  MoveL 8739 to (-32.14, 37, 125.68) mm, rotated rx -180 ry 0 rz 180 deg; joints [-169.099, 67.153, -85.949, 168.501, 71.555, 3.683]
  Call Extruder(466.13359)
  MoveL 8740 to (-31.9, 36.9, 125.68) mm, rotated rx 180 ry 0 rz 180 deg; joints [-169.115, 67.132, -85.961, 168.515, 71.522, 3.684]
  MoveL 8741 to (-31.9, 36.9, 125.68) mm, rotated rx 180 ry 0 rz 180 deg; joints [-169.115, 67.132, -85.961, 168.515, 71.522, 3.684]
  Call Extruder(466.29670)
  MoveL 8742 to (-31.64, 36.79, 125.68) mm, rotated rx 180 ry 0 rz 180 deg; joints [-169.132, 67.109, -85.974, 168.531, 71.486, 3.686]
  MoveL 8743 to (-31.64, 36.79, 125.68) mm, rotated rx 180 ry 0 rz 180 deg; joints [-169.132, 67.109, -85.974, 168.531, 71.486, 3.686]
  Call Extruder(466.41015)
  MoveL 8744 to (-31.45, 36.73, 125.68) mm, rotated rx -180 ry 0 rz 180 deg; joints [-169.139, 67.093, -85.983, 168.537, 71.461, 3.689]
  MoveL 8745 to (-31.45, 36.73, 125.68) mm, rotated rx -180 ry 0 rz 180 deg; joints [-169.139, 67.093, -85.983, 168.537, 71.461, 3.689]
  Call Extruder(466.52317)
  MoveL 8746 to (-31.26, 36.67, 125.68) mm, rotated rx -180 ry 0 rz -180 deg; joints [-169.146, 67.077, -85.992, 168.543, 71.435, 3.692]
  MoveL 8747 to (-31.26, 36.67, 125.68) mm, rotated rx -180 ry 0 rz -180 deg; joints [-169.146, 67.077, -85.992, 168.543, 71.435, 3.692]
  Call Extruder(466.63573)
  MoveL 8748 to (-31.07, 36.61, 125.68) mm, rotated rx -180 ry 0 rz -180 deg; joints [-169.154, 67.06, -86.001, 168.549, 71.41, 3.695]
  MoveL 8749 to (-31.07, 36.61, 125.68) mm, rotated rx -180 ry 0 rz -180 deg; joints [-169.154, 67.06, -86.001, 168.549, 71.41, 3.695]
  Call Extruder(466.74786)
  MoveL 8750 to (-30.88, 36.55, 125.68) mm, rotated rx 180 ry 0 rz -180 deg; joints [-169.161, 67.044, -86.01, 168.555, 71.385, 3.698]
  MoveL 8751 to (-30.88, 36.55, 125.68) mm, rotated rx 180 ry 0 rz -180 deg; joints [-169.161, 67.044, -86.01, 168.555, 71.385, 3.698]
  Call Extruder(466.85954)
  MoveL 8752 to (-30.7, 36.49, 125.68) mm, rotated rx -180 ry 0 rz -180 deg; joints [-169.168, 67.028, -86.019, 168.561, 71.36, 3.701]
  MoveL 8753 to (-30.7, 36.49, 125.68) mm, rotated rx -180 ry 0 rz -180 deg; joints [-169.168, 67.028, -86.019, 168.561, 71.36, 3.701]
  Call Extruder(466.99061)
  MoveL 8754 to (-30.47, 36.42, 125.68) mm, rotated rx -180 ry 0 rz -180 deg; joints [-169.175, 67.008, -86.03, 168.566, 71.33, 3.704]
  MoveL 8755 to (-30.47, 36.42, 125.68) mm, rotated rx -180 ry 0 rz -180 deg; joints [-169.175, 67.008, -86.03, 168.566, 71.33, 3.704]
  Call Extruder(467.12112)
  MoveL 8756 to (-30.25, 36.35, 125.68) mm, rotated rx -180 ry 0 rz -180 deg; joints [-169.182, 66.989, -86.04, 168.572, 71.3, 3.708]
  MoveL 8757 to (-30.25, 36.35, 125.68) mm, rotated rx -180 ry 0 rz -180 deg; joints [-169.182, 66.989, -86.04, 168.572, 71.3, 3.708]
  Call Extruder(467.25107)
  MoveL 8758 to (-30.02, 36.28, 125.68) mm, rotated rx -180 ry 0 rz -180 deg; joints [-169.19, 66.97, -86.051, 168.577, 71.27, 3.712]
  MoveL 8759 to (-30.02, 36.28, 125.68) mm, rotated rx -180 ry 0 rz -180 deg; joints [-169.19, 66.97, -86.051, 168.577, 71.27, 3.712]
  Call Extruder(467.38045)
  MoveL 8760 to (-29.8, 36.22, 125.68) mm, rotated rx 180 ry 0 rz -180 deg; joints [-169.197, 66.95, -86.061, 168.583, 71.24, 3.716]
  MoveL 8761 to (-29.8, 36.22, 125.68) mm, rotated rx 180 ry 0 rz -180 deg; joints [-169.197, 66.95, -86.061, 168.583, 71.24, 3.716]
  Call Extruder(467.50241)
  MoveL 8762 to (-29.59, 36.16, 125.68) mm, rotated rx 180 ry 0 rz 180 deg; joints [-169.202, 66.932, -86.071, 168.586, 71.212, 3.72]
  MoveL 8763 to (-29.59, 36.16, 125.68) mm, rotated rx 180 ry 0 rz 180 deg; joints [-169.202, 66.932, -86.071, 168.586, 71.212, 3.72]
  Call Extruder(467.61726)
  MoveL 8764 to (-29.38, 36.12, 125.68) mm, rotated rx -180 ry 0 rz -180 deg; joints [-169.203, 66.915, -86.081, 168.586, 71.186, 3.725]
  MoveL 8765 to (-29.38, 36.12, 125.68) mm, rotated rx -180 ry 0 rz -180 deg; joints [-169.203, 66.915, -86.081, 168.586, 71.186, 3.725]
  Call Extruder(467.73165)
  MoveL 8766 to (-29.18, 36.07, 125.68) mm, rotated rx 180 ry 0 rz 180 deg; joints [-169.205, 66.897, -86.09, 168.586, 71.16, 3.73]
  MoveL 8767 to (-29.18, 36.07, 125.68) mm, rotated rx 180 ry 0 rz 180 deg; joints [-169.205, 66.897, -86.09, 168.586, 71.16, 3.73]
  Call Extruder(467.84560)
  MoveL 8768 to (-28.97, 36.03, 125.68) mm, rotated rx 180 ry 0 rz -180 deg; joints [-169.207, 66.88, -86.099, 168.586, 71.133, 3.735]
  MoveL 8769 to (-28.97, 36.03, 125.68) mm, rotated rx 180 ry 0 rz -180 deg; joints [-169.207, 66.88, -86.099, 168.586, 71.133, 3.735]
  Call Extruder(467.95909)
  MoveL 8770 to (-28.77, 35.98, 125.68) mm, rotated rx -180 ry 0 rz -180 deg; joints [-169.208, 66.862, -86.109, 168.586, 71.107, 3.74]
  MoveL 8771 to (-28.77, 35.98, 125.68) mm, rotated rx -180 ry 0 rz -180 deg; joints [-169.208, 66.862, -86.109, 168.586, 71.107, 3.74]
  Call Extruder(468.09637)
  MoveL 8772 to (-28.52, 35.93, 125.68) mm, rotated rx 180 ry 0 rz -180 deg; joints [-169.209, 66.841, -86.12, 168.584, 71.075, 3.747]
  MoveL 8773 to (-28.52, 35.93, 125.68) mm, rotated rx 180 ry 0 rz -180 deg; joints [-169.209, 66.841, -86.12, 168.584, 71.075, 3.747]
  Call Extruder(468.23304)
  MoveL 8774 to (-28.27, 35.88, 125.68) mm, rotated rx -180 ry 0 rz 180 deg; joints [-169.209, 66.82, -86.132, 168.582, 71.043, 3.754]
  MoveL 8775 to (-28.27, 35.88, 125.68) mm, rotated rx -180 ry 0 rz 180 deg; joints [-169.209, 66.82, -86.132, 168.582, 71.043, 3.754]
  Call Extruder(468.36910)
  MoveL 8776 to (-28.02, 35.83, 125.68) mm, rotated rx -180 ry 0 rz -180 deg; joints [-169.21, 66.798, -86.143, 168.581, 71.011, 3.76]
  MoveL 8777 to (-28.02, 35.83, 125.68) mm, rotated rx -180 ry 0 rz -180 deg; joints [-169.21, 66.798, -86.143, 168.581, 71.011, 3.76]
  Call Extruder(468.50456)
  MoveL 8778 to (-27.77, 35.78, 125.68) mm, rotated rx -180 ry 0 rz -180 deg; joints [-169.21, 66.777, -86.154, 168.579, 70.979, 3.767]
  MoveL 8779 to (-27.77, 35.78, 125.68) mm, rotated rx -180 ry 0 rz -180 deg; joints [-169.21, 66.777, -86.154, 168.579, 70.979, 3.767]
  Call Extruder(468.63940)
  MoveL 8780 to (-27.52, 35.73, 125.68) mm, rotated rx -180 ry 0 rz 180 deg; joints [-169.211, 66.756, -86.166, 168.578, 70.947, 3.773]
  MoveL 8781 to (-27.52, 35.73, 125.68) mm, rotated rx -180 ry 0 rz 180 deg; joints [-169.211, 66.756, -86.166, 168.578, 70.947, 3.773]
  Call Extruder(468.77363)
  MoveL 8782 to (-27.28, 35.68, 125.68) mm, rotated rx -180 ry 0 rz 180 deg; joints [-169.212, 66.734, -86.177, 168.576, 70.915, 3.78]
  MoveL 8783 to (-27.28, 35.68, 125.68) mm, rotated rx -180 ry 0 rz 180 deg; joints [-169.212, 66.734, -86.177, 168.576, 70.915, 3.78]
  Call Extruder(468.90725)
  MoveL 8784 to (-27.03, 35.63, 125.68) mm, rotated rx 180 ry 0 rz 180 deg; joints [-169.212, 66.713, -86.188, 168.575, 70.883, 3.787]
  MoveL 8785 to (-27.03, 35.63, 125.68) mm, rotated rx 180 ry 0 rz 180 deg; joints [-169.212, 66.713, -86.188, 168.575, 70.883, 3.787]
  Call Extruder(469.06935)
  MoveL 8786 to (-26.72, 35.59, 125.68) mm, rotated rx 180 ry 0 rz 180 deg; joints [-169.21, 66.687, -86.202, 168.569, 70.844, 3.796]
  MoveL 8787 to (-26.72, 35.59, 125.68) mm, rotated rx 180 ry 0 rz 180 deg; joints [-169.21, 66.687, -86.202, 168.569, 70.844, 3.796]
  Call Extruder(469.23072)
  MoveL 8788 to (-26.41, 35.54, 125.68) mm, rotated rx -180 ry 0 rz 180 deg; joints [-169.207, 66.661, -86.215, 168.563, 70.805, 3.805]
  MoveL 8789 to (-26.41, 35.54, 125.68) mm, rotated rx -180 ry 0 rz 180 deg; joints [-169.207, 66.661, -86.215, 168.563, 70.805, 3.805]
  Call Extruder(469.39136)
  MoveL 8790 to (-26.11, 35.49, 125.68) mm, rotated rx 180 ry 0 rz 180 deg; joints [-169.204, 66.635, -86.229, 168.557, 70.767, 3.815]
  MoveL 8791 to (-26.11, 35.49, 125.68) mm, rotated rx 180 ry 0 rz 180 deg; joints [-169.204, 66.635, -86.229, 168.557, 70.767, 3.815]
  Call Extruder(469.55127)
  MoveL 8792 to (-25.8, 35.44, 125.68) mm, rotated rx 180 ry 0 rz 180 deg; joints [-169.201, 66.609, -86.242, 168.551, 70.728, 3.824]
  MoveL 8793 to (-25.8, 35.44, 125.68) mm, rotated rx 180 ry 0 rz 180 deg; joints [-169.201, 66.609, -86.242, 168.551, 70.728, 3.824]
  Call Extruder(469.71046)
  MoveL 8794 to (-25.5, 35.39, 125.68) mm, rotated rx -180 ry 0 rz -180 deg; joints [-169.198, 66.582, -86.256, 168.546, 70.689, 3.833]
  MoveL 8795 to (-25.5, 35.39, 125.68) mm, rotated rx -180 ry 0 rz -180 deg; joints [-169.198, 66.582, -86.256, 168.546, 70.689, 3.833]
  Call Extruder(469.86892)
  MoveL 8796 to (-25.19, 35.34, 125.68) mm, rotated rx -180 ry 0 rz -180 deg; joints [-169.195, 66.556, -86.269, 168.54, 70.65, 3.843]
  MoveL 8797 to (-25.19, 35.34, 125.68) mm, rotated rx -180 ry 0 rz -180 deg; joints [-169.195, 66.556, -86.269, 168.54, 70.65, 3.843]
  Call Extruder(470.06779)
  MoveL 8798 to (-24.8, 35.3, 125.68) mm, rotated rx 180 ry 0 rz 180 deg; joints [-169.187, 66.523, -86.286, 168.527, 70.602, 3.856]
  MoveL 8799 to (-24.8, 35.3, 125.68) mm, rotated rx 180 ry 0 rz 180 deg; joints [-169.187, 66.523, -86.286, 168.527, 70.602, 3.856]
  Call Extruder(470.26580)
  MoveL 8800 to (-24.42, 35.25, 125.68) mm, rotated rx -180 ry 0 rz -180 deg; joints [-169.178, 66.49, -86.303, 168.515, 70.554, 3.87]
  MoveL 8801 to (-24.42, 35.25, 125.68) mm, rotated rx -180 ry 0 rz -180 deg; joints [-169.178, 66.49, -86.303, 168.515, 70.554, 3.87]
  Call Extruder(470.46294)
  MoveL 8802 to (-24.03, 35.21, 125.68) mm, rotated rx -180 ry 0 rz -180 deg; joints [-169.17, 66.457, -86.32, 168.502, 70.506, 3.883]
  MoveL 8803 to (-24.03, 35.21, 125.68) mm, rotated rx -180 ry 0 rz -180 deg; joints [-169.17, 66.457, -86.32, 168.502, 70.506, 3.883]
  Call Extruder(470.65922)
  MoveL 8804 to (-23.64, 35.16, 125.68) mm, rotated rx -180 ry 0 rz 180 deg; joints [-169.161, 66.424, -86.337, 168.49, 70.457, 3.897]
  MoveL 8805 to (-23.64, 35.16, 125.68) mm, rotated rx -180 ry 0 rz 180 deg; joints [-169.161, 66.424, -86.337, 168.49, 70.457, 3.897]
  Call Extruder(470.90490)
  MoveL 8806 to (-23.15, 35.11, 125.68) mm, rotated rx 180 ry 0 rz 180 deg; joints [-169.147, 66.382, -86.357, 168.47, 70.397, 3.915]
  MoveL 8807 to (-23.15, 35.11, 125.68) mm, rotated rx 180 ry 0 rz 180 deg; joints [-169.147, 66.382, -86.357, 168.47, 70.397, 3.915]
  Call Extruder(471.19963)
  MoveL 8808 to (-22.56, 35.07, 125.68) mm, rotated rx 180 ry 0 rz 180 deg; joints [-169.127, 66.332, -86.382, 168.444, 70.325, 3.938]
  MoveL 8809 to (-22.56, 35.07, 125.68) mm, rotated rx 180 ry 0 rz 180 deg; joints [-169.127, 66.332, -86.382, 168.444, 70.325, 3.938]
  Call Extruder(471.49303)
  MoveL 8810 to (-21.97, 35.02, 125.68) mm, rotated rx -180 ry 0 rz -180 deg; joints [-169.107, 66.282, -86.407, 168.417, 70.252, 3.962]
  MoveL 8811 to (-21.97, 35.02, 125.68) mm, rotated rx -180 ry 0 rz -180 deg; joints [-169.107, 66.282, -86.407, 168.417, 70.252, 3.962]
  Call Extruder(471.92636)
  MoveL 8812 to (-21.1, 34.98, 125.68) mm, rotated rx 180 ry 0 rz -180 deg; joints [-169.069, 66.207, -86.444, 168.369, 70.146, 3.999]
  MoveL 8813 to (-21.1, 34.98, 125.68) mm, rotated rx 180 ry 0 rz -180 deg; joints [-169.069, 66.207, -86.444, 168.369, 70.146, 3.999]
  Call Extruder(472.49852)
  MoveL 8814 to (-19.94, 34.93, 125.68) mm, rotated rx -180 ry 0 rz -180 deg; joints [-169.014, 66.108, -86.492, 168.3, 70.006, 4.05]
  MoveL 8815 to (-19.94, 34.93, 125.68) mm, rotated rx -180 ry 0 rz -180 deg; joints [-169.014, 66.108, -86.492, 168.3, 70.006, 4.05]
  Call Extruder(472.92635)
  MoveL 8816 to (-19.06, 34.91, 125.68) mm, rotated rx -180 ry 0 rz -180 deg; joints [-168.967, 66.034, -86.527, 168.242, 69.901, 4.091]
  Call Extruder(589.57504)
  MoveL 8817 to (219.06, 34.91, 125.68) mm, rotated rx -180 ry 0 rz 180 deg; joints [-30.588, 54.353, -88.738, 35.613, 119.089, 19.2]
  MoveL 8818 to (219.06, 34.91, 125.68) mm, rotated rx -180 ry 0 rz 180 deg; joints [-30.588, 54.353, -88.738, 35.613, 119.089, 19.2]
  Call Extruder(590.29061)
  MoveL 8819 to (220.52, 34.95, 125.68) mm, rotated rx -180 ry 0 rz 180 deg; joints [-30.009, 54.502, -88.741, 34.939, 119.158, 18.798]
  MoveL 8820 to (220.52, 34.95, 125.68) mm, rotated rx -180 ry 0 rz 180 deg; joints [-30.009, 54.502, -88.741, 34.939, 119.158, 18.798]
  Call Extruder(590.86535)
  MoveL 8821 to (221.68, 35, 125.68) mm, rotated rx -180 ry 0 rz 180 deg; joints [-29.572, 54.622, -88.743, 34.427, 119.201, 18.489]
  MoveL 8822 to (221.68, 35, 125.68) mm, rotated rx -180 ry 0 rz 180 deg; joints [-29.572, 54.622, -88.743, 34.427, 119.201, 18.489]
  Call Extruder(591.15874)
  MoveL 8823 to (222.27, 35.05, 125.68) mm, rotated rx -180 ry 0 rz 180 deg; joints [-29.371, 54.685, -88.744, 34.19, 119.213, 18.343]
  MoveL 8824 to (222.27, 35.05, 125.68) mm, rotated rx -180 ry 0 rz 180 deg; joints [-29.371, 54.685, -88.744, 34.19, 119.213, 18.343]
  Call Extruder(591.45347)
  MoveL 8825 to (222.86, 35.09, 125.68) mm, rotated rx -180 ry 0 rz 180 deg; joints [-29.173, 54.747, -88.744, 33.955, 119.224, 18.198]
  MoveL 8826 to (222.86, 35.09, 125.68) mm, rotated rx -180 ry 0 rz 180 deg; joints [-29.173, 54.747, -88.744, 33.955, 119.224, 18.198]
  Call Extruder(591.74952)
  MoveL 8827 to (223.45, 35.14, 125.68) mm, rotated rx -180 ry 0 rz 180 deg; joints [-28.978, 54.809, -88.745, 33.723, 119.233, 18.055]
  MoveL 8828 to (223.45, 35.14, 125.68) mm, rotated rx -180 ry 0 rz 180 deg; joints [-28.978, 54.809, -88.745, 33.723, 119.233, 18.055]
  Call Extruder(591.94580)
  MoveL 8829 to (223.83, 35.18, 125.68) mm, rotated rx -180 ry 0 rz 180 deg; joints [-28.862, 54.851, -88.745, 33.584, 119.235, 17.967]
  MoveL 8830 to (223.83, 35.18, 125.68) mm, rotated rx -180 ry 0 rz 180 deg; joints [-28.862, 54.851, -88.745, 33.584, 119.235, 17.967]
  Call Extruder(592.14294)
  MoveL 8831 to (224.22, 35.23, 125.68) mm, rotated rx -180 ry 0 rz 180 deg; joints [-28.747, 54.893, -88.745, 33.445, 119.235, 17.879]
  MoveL 8832 to (224.22, 35.23, 125.68) mm, rotated rx -180 ry 0 rz 180 deg; joints [-28.747, 54.893, -88.745, 33.445, 119.235, 17.879]
  Call Extruder(592.34095)
  MoveL 8833 to (224.61, 35.27, 125.68) mm, rotated rx -180 ry 0 rz 180 deg; joints [-28.633, 54.935, -88.746, 33.309, 119.235, 17.793]
  MoveL 8834 to (224.61, 35.27, 125.68) mm, rotated rx -180 ry 0 rz 180 deg; joints [-28.633, 54.935, -88.746, 33.309, 119.235, 17.793]
  Call Extruder(592.53982)
  MoveL 8835 to (225, 35.32, 125.68) mm, rotated rx 180 ry 0 rz 180 deg; joints [-28.52, 54.977, -88.746, 33.173, 119.235, 17.706]
  MoveL 8836 to (225, 35.32, 125.68) mm, rotated rx 180 ry 0 rz 180 deg; joints [-28.52, 54.977, -88.746, 33.173, 119.235, 17.706]
  Call Extruder(592.71890)
  MoveL 8837 to (225.34, 35.37, 125.68) mm, rotated rx -180 ry 0 rz 180 deg; joints [-28.425, 55.015, -88.746, 33.057, 119.232, 17.632]
  MoveL 8838 to (225.34, 35.37, 125.68) mm, rotated rx -180 ry 0 rz 180 deg; joints [-28.425, 55.015, -88.746, 33.057, 119.232, 17.632]
  Call Extruder(592.87809)
  MoveL 8839 to (225.65, 35.42, 125.68) mm, rotated rx 180 ry 0 rz 180 deg; joints [-28.346, 55.049, -88.746, 32.961, 119.228, 17.569]
  MoveL 8840 to (225.65, 35.42, 125.68) mm, rotated rx 180 ry 0 rz 180 deg; joints [-28.346, 55.049, -88.746, 32.961, 119.228, 17.569]
  Call Extruder(593.03800)
  MoveL 8841 to (225.96, 35.47, 125.68) mm, rotated rx -180 ry 0 rz 180 deg; joints [-28.267, 55.082, -88.746, 32.864, 119.223, 17.506]
  MoveL 8842 to (225.96, 35.47, 125.68) mm, rotated rx -180 ry 0 rz 180 deg; joints [-28.267, 55.082, -88.746, 32.864, 119.223, 17.506]
  Call Extruder(593.19864)
  MoveL 8843 to (226.26, 35.51, 125.68) mm, rotated rx -180 ry 0 rz 180 deg; joints [-28.19, 55.116, -88.746, 32.77, 119.218, 17.443]
  MoveL 8844 to (226.26, 35.51, 125.68) mm, rotated rx -180 ry 0 rz 180 deg; joints [-28.19, 55.116, -88.746, 32.77, 119.218, 17.443]
  Call Extruder(593.36001)
  MoveL 8845 to (226.57, 35.56, 125.68) mm, rotated rx -180 ry 0 rz -180 deg; joints [-28.112, 55.15, -88.746, 32.675, 119.213, 17.381]
  MoveL 8846 to (226.57, 35.56, 125.68) mm, rotated rx -180 ry 0 rz -180 deg; joints [-28.112, 55.15, -88.746, 32.675, 119.213, 17.381]
  Call Extruder(593.52210)
  MoveL 8847 to (226.87, 35.61, 125.68) mm, rotated rx -180 ry 0 rz 180 deg; joints [-28.036, 55.184, -88.746, 32.581, 119.207, 17.319]
  MoveL 8848 to (226.87, 35.61, 125.68) mm, rotated rx -180 ry 0 rz 180 deg; joints [-28.036, 55.184, -88.746, 32.581, 119.207, 17.319]
  Call Extruder(593.67030)
  MoveL 8849 to (227.15, 35.66, 125.68) mm, rotated rx 180 ry 0 rz 180 deg; joints [-27.971, 55.215, -88.746, 32.5, 119.2, 17.265]
  MoveL 8850 to (227.15, 35.66, 125.68) mm, rotated rx 180 ry 0 rz 180 deg; joints [-27.971, 55.215, -88.746, 32.5, 119.2, 17.265]
  Call Extruder(593.80453)
  MoveL 8851 to (227.4, 35.71, 125.68) mm, rotated rx -180 ry 0 rz 180 deg; joints [-27.915, 55.243, -88.746, 32.431, 119.193, 17.219]
  MoveL 8852 to (227.4, 35.71, 125.68) mm, rotated rx -180 ry 0 rz 180 deg; joints [-27.915, 55.243, -88.746, 32.431, 119.193, 17.219]
  Call Extruder(593.93938)
  MoveL 8853 to (227.65, 35.76, 125.68) mm, rotated rx -180 ry 0 rz -180 deg; joints [-27.861, 55.271, -88.746, 32.363, 119.185, 17.172]
  MoveL 8854 to (227.65, 35.76, 125.68) mm, rotated rx -180 ry 0 rz -180 deg; joints [-27.861, 55.271, -88.746, 32.363, 119.185, 17.172]
  Call Extruder(594.07483)
  MoveL 8855 to (227.9, 35.81, 125.68) mm, rotated rx -180 ry 0 rz 180 deg; joints [-27.807, 55.299, -88.745, 32.295, 119.178, 17.126]
  MoveL 8856 to (227.9, 35.81, 125.68) mm, rotated rx -180 ry 0 rz 180 deg; joints [-27.807, 55.299, -88.745, 32.295, 119.178, 17.126]
  Call Extruder(594.21089)
  MoveL 8857 to (228.15, 35.86, 125.68) mm, rotated rx 180 ry 0 rz 180 deg; joints [-27.753, 55.327, -88.745, 32.228, 119.169, 17.08]
  MoveL 8858 to (228.15, 35.86, 125.68) mm, rotated rx 180 ry 0 rz 180 deg; joints [-27.753, 55.327, -88.745, 32.228, 119.169, 17.08]
  Call Extruder(594.34757)
  MoveL 8859 to (228.4, 35.91, 125.68) mm, rotated rx 180 ry 0 rz 180 deg; joints [-27.699, 55.355, -88.745, 32.161, 119.161, 17.034]
  MoveL 8860 to (228.4, 35.91, 125.68) mm, rotated rx 180 ry 0 rz 180 deg; joints [-27.699, 55.355, -88.745, 32.161, 119.161, 17.034]
  Call Extruder(594.48485)
  MoveL 8861 to (228.64, 35.96, 125.68) mm, rotated rx -180 ry 0 rz -180 deg; joints [-27.646, 55.383, -88.745, 32.094, 119.153, 16.989]
  MoveL 8862 to (228.64, 35.96, 125.68) mm, rotated rx -180 ry 0 rz -180 deg; joints [-27.646, 55.383, -88.745, 32.094, 119.153, 16.989]
  Call Extruder(594.61052)
  MoveL 8863 to (228.87, 36, 125.68) mm, rotated rx 180 ry 0 rz 180 deg; joints [-27.599, 55.408, -88.745, 32.036, 119.145, 16.948]
  MoveL 8864 to (228.87, 36, 125.68) mm, rotated rx 180 ry 0 rz 180 deg; joints [-27.599, 55.408, -88.745, 32.036, 119.145, 16.948]
  Call Extruder(594.72447)
  MoveL 8865 to (229.08, 36.05, 125.68) mm, rotated rx -180 ry 0 rz 180 deg; joints [-27.559, 55.431, -88.744, 31.984, 119.137, 16.912]
  MoveL 8866 to (229.08, 36.05, 125.68) mm, rotated rx -180 ry 0 rz 180 deg; joints [-27.559, 55.431, -88.744, 31.984, 119.137, 16.912]
  Call Extruder(594.83887)
  MoveL 8867 to (229.28, 36.09, 125.68) mm, rotated rx -180 ry 0 rz 180 deg; joints [-27.518, 55.455, -88.744, 31.933, 119.129, 16.877]
  MoveL 8868 to (229.28, 36.09, 125.68) mm, rotated rx -180 ry 0 rz 180 deg; joints [-27.518, 55.455, -88.744, 31.933, 119.129, 16.877]
  Call Extruder(594.95372)
  MoveL 8869 to (229.48, 36.14, 125.68) mm, rotated rx -180 ry 0 rz 180 deg; joints [-27.479, 55.478, -88.744, 31.882, 119.12, 16.841]
  MoveL 8870 to (229.48, 36.14, 125.68) mm, rotated rx -180 ry 0 rz 180 deg; joints [-27.479, 55.478, -88.744, 31.882, 119.12, 16.841]
  Call Extruder(595.06902)
  MoveL 8871 to (229.69, 36.18, 125.68) mm, rotated rx -180 ry 0 rz 180 deg; joints [-27.439, 55.501, -88.744, 31.832, 119.112, 16.806]
  MoveL 8872 to (229.69, 36.18, 125.68) mm, rotated rx -180 ry 0 rz 180 deg; joints [-27.439, 55.501, -88.744, 31.832, 119.112, 16.806]
  Call Extruder(595.20041)
  MoveL 8873 to (229.92, 36.25, 125.68) mm, rotated rx -180 ry 0 rz 180 deg; joints [-27.404, 55.528, -88.743, 31.786, 119.099, 16.771]
  MoveL 8874 to (229.92, 36.25, 125.68) mm, rotated rx -180 ry 0 rz 180 deg; joints [-27.404, 55.528, -88.743, 31.786, 119.099, 16.771]
  Call Extruder(595.31352)
  MoveL 8875 to (230.11, 36.31, 125.68) mm, rotated rx -180 ry 0 rz 180 deg; joints [-27.377, 55.55, -88.743, 31.75, 119.087, 16.743]
  MoveL 8876 to (230.11, 36.31, 125.68) mm, rotated rx -180 ry 0 rz 180 deg; joints [-27.377, 55.55, -88.743, 31.75, 119.087, 16.743]
  Call Extruder(595.42707)
  MoveL 8877 to (230.31, 36.37, 125.68) mm, rotated rx -180 ry 0 rz 180 deg; joints [-27.351, 55.573, -88.743, 31.714, 119.075, 16.715]
  MoveL 8878 to (230.31, 36.37, 125.68) mm, rotated rx -180 ry 0 rz 180 deg; joints [-27.351, 55.573, -88.743, 31.714, 119.075, 16.715]
  Call Extruder(595.54106)
  MoveL 8879 to (230.5, 36.43, 125.68) mm, rotated rx -180 ry 0 rz 180 deg; joints [-27.325, 55.596, -88.742, 31.679, 119.062, 16.687]
  MoveL 8880 to (230.5, 36.43, 125.68) mm, rotated rx -180 ry 0 rz 180 deg; joints [-27.325, 55.596, -88.742, 31.679, 119.062, 16.687]
  Call Extruder(595.65549)
  MoveL 8881 to (230.7, 36.49, 125.68) mm, rotated rx -180 ry 0 rz 180 deg; joints [-27.299, 55.619, -88.742, 31.644, 119.05, 16.659]
  MoveL 8882 to (230.7, 36.49, 125.68) mm, rotated rx -180 ry 0 rz 180 deg; joints [-27.299, 55.619, -88.742, 31.644, 119.05, 16.659]
  Call Extruder(595.76739)
  MoveL 8883 to (230.88, 36.55, 125.68) mm, rotated rx 180 ry 0 rz 180 deg; joints [-27.276, 55.642, -88.742, 31.612, 119.037, 16.633]
  MoveL 8884 to (230.88, 36.55, 125.68) mm, rotated rx 180 ry 0 rz 180 deg; joints [-27.276, 55.642, -88.742, 31.612, 119.037, 16.633]
  Call Extruder(595.87973)
  MoveL 8885 to (231.07, 36.61, 125.68) mm, rotated rx -180 ry 0 rz 180 deg; joints [-27.253, 55.664, -88.741, 31.58, 119.025, 16.607]
  MoveL 8886 to (231.07, 36.61, 125.68) mm, rotated rx -180 ry 0 rz 180 deg; joints [-27.253, 55.664, -88.741, 31.58, 119.025, 16.607]
  Call Extruder(595.99252)
  MoveL 8887 to (231.26, 36.67, 125.68) mm, rotated rx -180 ry 0 rz -180 deg; joints [-27.231, 55.686, -88.741, 31.549, 119.012, 16.582]
  MoveL 8888 to (231.26, 36.67, 125.68) mm, rotated rx -180 ry 0 rz -180 deg; joints [-27.231, 55.686, -88.741, 31.549, 119.012, 16.582]
  Call Extruder(596.10575)
  MoveL 8889 to (231.45, 36.73, 125.68) mm, rotated rx -180 ry 0 rz 180 deg; joints [-27.208, 55.709, -88.74, 31.517, 118.999, 16.556]
  MoveL 8890 to (231.45, 36.73, 125.68) mm, rotated rx -180 ry 0 rz 180 deg; joints [-27.208, 55.709, -88.74, 31.517, 118.999, 16.556]
  Call Extruder(596.21943)
  MoveL 8891 to (231.64, 36.79, 125.68) mm, rotated rx -180 ry 0 rz 180 deg; joints [-27.185, 55.731, -88.74, 31.486, 118.986, 16.531]
  MoveL 8892 to (231.64, 36.79, 125.68) mm, rotated rx -180 ry 0 rz 180 deg; joints [-27.185, 55.731, -88.74, 31.486, 118.986, 16.531]
  Call Extruder(596.40139)
  MoveL 8893 to (231.93, 36.91, 125.68) mm, rotated rx -180 ry 0 rz 180 deg; joints [-27.167, 55.767, -88.739, 31.455, 118.96, 16.499]
  MoveL 8894 to (231.93, 36.91, 125.68) mm, rotated rx -180 ry 0 rz 180 deg; joints [-27.167, 55.767, -88.739, 31.455, 118.96, 16.499]
  Call Extruder(596.58411)
  MoveL 8895 to (232.22, 37.04, 125.68) mm, rotated rx 180 ry 0 rz -180 deg; joints [-27.149, 55.803, -88.739, 31.425, 118.933, 16.468]
  MoveL 8896 to (232.22, 37.04, 125.68) mm, rotated rx 180 ry 0 rz -180 deg; joints [-27.149, 55.803, -88.739, 31.425, 118.933, 16.468]
  Call Extruder(596.75452)
  MoveL 8897 to (232.49, 37.15, 125.68) mm, rotated rx 180 ry 0 rz 180 deg; joints [-27.133, 55.836, -88.738, 31.398, 118.909, 16.439]
  MoveL 8898 to (232.49, 37.15, 125.68) mm, rotated rx 180 ry 0 rz 180 deg; joints [-27.133, 55.836, -88.738, 31.398, 118.909, 16.439]
  Call Extruder(596.91252)
  MoveL 8899 to (232.74, 37.26, 125.68) mm, rotated rx 180 ry 0 rz 180 deg; joints [-27.121, 55.867, -88.737, 31.375, 118.885, 16.414]
  MoveL 8900 to (232.74, 37.26, 125.68) mm, rotated rx 180 ry 0 rz 180 deg; joints [-27.121, 55.867, -88.737, 31.375, 118.885, 16.414]
  Call Extruder(597.07112)
  MoveL 8901 to (232.99, 37.36, 125.68) mm, rotated rx -180 ry 0 rz -180 deg; joints [-27.108, 55.898, -88.737, 31.352, 118.862, 16.388]
  MoveL 8902 to (232.99, 37.36, 125.68) mm, rotated rx -180 ry 0 rz -180 deg; joints [-27.108, 55.898, -88.737, 31.352, 118.862, 16.388]
  Call Extruder(597.27729)
  MoveL 8903 to (233.29, 37.54, 125.68) mm, rotated rx 180 ry 0 rz 180 deg; joints [-27.12, 55.938, -88.736, 31.353, 118.824, 16.37]
  MoveL 8904 to (233.29, 37.54, 125.68) mm, rotated rx 180 ry 0 rz 180 deg; joints [-27.12, 55.938, -88.736, 31.353, 118.824, 16.37]
  Call Extruder(597.48423)
  MoveL 8905 to (233.6, 37.71, 125.68) mm, rotated rx 180 ry 0 rz -180 deg; joints [-27.132, 55.978, -88.735, 31.355, 118.785, 16.352]
  MoveL 8906 to (233.6, 37.71, 125.68) mm, rotated rx 180 ry 0 rz -180 deg; joints [-27.132, 55.978, -88.735, 31.355, 118.785, 16.352]
  Call Extruder(597.69196)
  MoveL 8907 to (233.9, 37.89, 125.68) mm, rotated rx 180 ry 0 rz 180 deg; joints [-27.144, 56.018, -88.733, 31.356, 118.747, 16.334]
  MoveL 8908 to (233.9, 37.89, 125.68) mm, rotated rx 180 ry 0 rz 180 deg; joints [-27.144, 56.018, -88.733, 31.356, 118.747, 16.334]
  Call Extruder(597.90046)
  MoveL 8909 to (234.21, 38.07, 125.68) mm, rotated rx -180 ry 0 rz 180 deg; joints [-27.156, 56.058, -88.732, 31.358, 118.709, 16.316]
  MoveL 8910 to (234.21, 38.07, 125.68) mm, rotated rx -180 ry 0 rz 180 deg; joints [-27.156, 56.058, -88.732, 31.358, 118.709, 16.316]
  Call Extruder(598.08001)
  MoveL 8911 to (234.45, 38.24, 125.68) mm, rotated rx -180 ry 0 rz 180 deg; joints [-27.187, 56.092, -88.731, 31.382, 118.67, 16.312]
  MoveL 8912 to (234.45, 38.24, 125.68) mm, rotated rx -180 ry 0 rz 180 deg; joints [-27.187, 56.092, -88.731, 31.382, 118.67, 16.312]
  Call Extruder(598.41342)
  MoveL 8913 to (234.9, 38.57, 125.68) mm, rotated rx 180 ry 0 rz 180 deg; joints [-27.245, 56.154, -88.729, 31.427, 118.599, 16.304]
  MoveL 8914 to (234.9, 38.57, 125.68) mm, rotated rx 180 ry 0 rz 180 deg; joints [-27.245, 56.154, -88.729, 31.427, 118.599, 16.304]
  Call Extruder(598.74802)
  MoveL 8915 to (235.35, 38.9, 125.68) mm, rotated rx -180 ry 0 rz 180 deg; joints [-27.302, 56.217, -88.727, 31.471, 118.528, 16.296]
  Call Extruder(599.57597)
  MoveL 8916 to (236.39, 39.81, 125.68) mm, rotated rx 180 ry 0 rz 180 deg; joints [-27.525, 56.368, -88.722, 31.67, 118.332, 16.318]
  Call Extruder(600.40391)
  MoveL 8917 to (237.3, 40.85, 125.68) mm, rotated rx -180 ry 0 rz 180 deg; joints [-27.851, 56.514, -88.716, 31.983, 118.111, 16.395]
  Call Extruder(600.57121)
  MoveL 8918 to (237.47, 41.07, 125.68) mm, rotated rx 180 ry 0 rz 180 deg; joints [-27.932, 56.542, -88.715, 32.062, 118.063, 16.419]
  MoveL 8919 to (237.47, 41.07, 125.68) mm, rotated rx 180 ry 0 rz 180 deg; joints [-27.932, 56.542, -88.715, 32.062, 118.063, 16.419]
  Call Extruder(600.90463)
  MoveL 8920 to (237.79, 41.52, 125.68) mm, rotated rx 180 ry 0 rz -180 deg; joints [-28.091, 56.598, -88.712, 32.218, 117.968, 16.465]
  MoveL 8921 to (237.79, 41.52, 125.68) mm, rotated rx 180 ry 0 rz -180 deg; joints [-28.091, 56.598, -88.712, 32.218, 117.968, 16.465]
  Call Extruder(601.23686)
  MoveL 8922 to (238.12, 41.98, 125.68) mm, rotated rx -180 ry 0 rz -180 deg; joints [-28.249, 56.655, -88.71, 32.372, 117.874, 16.509]
  MoveL 8923 to (238.12, 41.98, 125.68) mm, rotated rx -180 ry 0 rz -180 deg; joints [-28.249, 56.655, -88.71, 32.372, 117.874, 16.509]
  Call Extruder(601.35455)
  MoveL 8924 to (238.22, 42.15, 125.68) mm, rotated rx -180 ry 0 rz 180 deg; joints [-28.315, 56.674, -88.709, 32.439, 117.838, 16.531]
  MoveL 8925 to (238.22, 42.15, 125.68) mm, rotated rx -180 ry 0 rz 180 deg; joints [-28.315, 56.674, -88.709, 32.439, 117.838, 16.531]
  Call Extruder(601.56228)
  MoveL 8926 to (238.4, 42.45, 125.68) mm, rotated rx -180 ry 0 rz 180 deg; joints [-28.434, 56.707, -88.707, 32.557, 117.775, 16.569]
  MoveL 8927 to (238.4, 42.45, 125.68) mm, rotated rx -180 ry 0 rz 180 deg; joints [-28.434, 56.707, -88.707, 32.557, 117.775, 16.569]
  Call Extruder(601.76922)
  MoveL 8928 to (238.57, 42.75, 125.68) mm, rotated rx -180 ry 0 rz 180 deg; joints [-28.552, 56.741, -88.706, 32.675, 117.711, 16.607]
  MoveL 8929 to (238.57, 42.75, 125.68) mm, rotated rx -180 ry 0 rz 180 deg; joints [-28.552, 56.741, -88.706, 32.675, 117.711, 16.607]
  Call Extruder(601.97539)
  MoveL 8930 to (238.75, 43.06, 125.68) mm, rotated rx 180 ry 0 rz 180 deg; joints [-28.669, 56.774, -88.704, 32.792, 117.648, 16.644]
  MoveL 8931 to (238.75, 43.06, 125.68) mm, rotated rx 180 ry 0 rz 180 deg; joints [-28.669, 56.774, -88.704, 32.792, 117.648, 16.644]
  Call Extruder(602.15708)
  MoveL 8932 to (238.89, 43.33, 125.68) mm, rotated rx -180 ry 0 rz 180 deg; joints [-28.78, 56.803, -88.703, 32.903, 117.591, 16.682]
  MoveL 8933 to (238.89, 43.33, 125.68) mm, rotated rx -180 ry 0 rz 180 deg; joints [-28.78, 56.803, -88.703, 32.903, 117.591, 16.682]
  Call Extruder(602.31509)
  MoveL 8934 to (239, 43.58, 125.68) mm, rotated rx -180 ry 0 rz -180 deg; joints [-28.886, 56.827, -88.701, 33.011, 117.539, 16.719]
  MoveL 8935 to (239, 43.58, 125.68) mm, rotated rx -180 ry 0 rz -180 deg; joints [-28.886, 56.827, -88.701, 33.011, 117.539, 16.719]
  Call Extruder(602.47250)
  MoveL 8936 to (239.1, 43.83, 125.68) mm, rotated rx -180 ry 0 rz 180 deg; joints [-28.991, 56.851, -88.7, 33.117, 117.488, 16.756]
  MoveL 8937 to (239.1, 43.83, 125.68) mm, rotated rx -180 ry 0 rz 180 deg; joints [-28.991, 56.851, -88.7, 33.117, 117.488, 16.756]
  Call Extruder(602.65521)
  MoveL 8938 to (239.23, 44.12, 125.68) mm, rotated rx -180 ry 0 rz 180 deg; joints [-29.116, 56.879, -88.699, 33.244, 117.427, 16.8]
  MoveL 8939 to (239.23, 44.12, 125.68) mm, rotated rx -180 ry 0 rz 180 deg; joints [-29.116, 56.879, -88.699, 33.244, 117.427, 16.8]
  Call Extruder(602.83717)
  MoveL 8940 to (239.35, 44.42, 125.68) mm, rotated rx 180 ry 0 rz 180 deg; joints [-29.24, 56.907, -88.697, 33.369, 117.367, 16.844]
  MoveL 8941 to (239.35, 44.42, 125.68) mm, rotated rx 180 ry 0 rz 180 deg; joints [-29.24, 56.907, -88.697, 33.369, 117.367, 16.844]
  Call Extruder(602.98450)
  MoveL 8942 to (239.44, 44.66, 125.68) mm, rotated rx -180 ry 0 rz -180 deg; joints [-29.343, 56.929, -88.696, 33.474, 117.318, 16.88]
  MoveL 8943 to (239.44, 44.66, 125.68) mm, rotated rx -180 ry 0 rz -180 deg; joints [-29.343, 56.929, -88.696, 33.474, 117.318, 16.88]
  Call Extruder(603.09774)
  MoveL 8944 to (239.5, 44.85, 125.68) mm, rotated rx -180 ry 0 rz 180 deg; joints [-29.428, 56.945, -88.695, 33.56, 117.279, 16.911]
  MoveL 8945 to (239.5, 44.85, 125.68) mm, rotated rx -180 ry 0 rz 180 deg; joints [-29.428, 56.945, -88.695, 33.56, 117.279, 16.911]
  Call Extruder(603.21053)
  MoveL 8946 to (239.56, 45.03, 125.68) mm, rotated rx -180 ry 0 rz -180 deg; joints [-29.512, 56.961, -88.694, 33.645, 117.24, 16.942]
  MoveL 8947 to (239.56, 45.03, 125.68) mm, rotated rx -180 ry 0 rz -180 deg; joints [-29.512, 56.961, -88.694, 33.645, 117.24, 16.942]
  Call Extruder(603.32287)
  MoveL 8948 to (239.62, 45.22, 125.68) mm, rotated rx -180 ry 0 rz 180 deg; joints [-29.596, 56.978, -88.693, 33.73, 117.201, 16.973]
  MoveL 8949 to (239.62, 45.22, 125.68) mm, rotated rx -180 ry 0 rz 180 deg; joints [-29.596, 56.978, -88.693, 33.73, 117.201, 16.973]
  Call Extruder(603.43477)
  MoveL 8950 to (239.68, 45.41, 125.68) mm, rotated rx 180 ry 0 rz -180 deg; joints [-29.679, 56.994, -88.692, 33.815, 117.162, 17.003]
  MoveL 8951 to (239.68, 45.41, 125.68) mm, rotated rx 180 ry 0 rz -180 deg; joints [-29.679, 56.994, -88.692, 33.815, 117.162, 17.003]
  Call Extruder(603.55618)
  MoveL 8952 to (239.75, 45.62, 125.68) mm, rotated rx -180 ry 0 rz 180 deg; joints [-29.77, 57.012, -88.691, 33.908, 117.12, 17.036]
  MoveL 8953 to (239.75, 45.62, 125.68) mm, rotated rx -180 ry 0 rz 180 deg; joints [-29.77, 57.012, -88.691, 33.908, 117.12, 17.036]
  Call Extruder(603.68697)
  MoveL 8954 to (239.82, 45.84, 125.68) mm, rotated rx -180 ry 0 rz 180 deg; joints [-29.871, 57.031, -88.69, 34.01, 117.074, 17.072]
  MoveL 8955 to (239.82, 45.84, 125.68) mm, rotated rx -180 ry 0 rz 180 deg; joints [-29.871, 57.031, -88.69, 34.01, 117.074, 17.072]
  Call Extruder(603.81719)
  MoveL 8956 to (239.88, 46.06, 125.68) mm, rotated rx -180 ry 0 rz 180 deg; joints [-29.97, 57.049, -88.689, 34.111, 117.028, 17.108]
  MoveL 8957 to (239.88, 46.06, 125.68) mm, rotated rx -180 ry 0 rz 180 deg; joints [-29.97, 57.049, -88.689, 34.111, 117.028, 17.108]
  Call Extruder(603.94685)
  MoveL 8958 to (239.95, 46.29, 125.68) mm, rotated rx -180 ry 0 rz 180 deg; joints [-30.069, 57.069, -88.688, 34.211, 116.982, 17.144]
  MoveL 8959 to (239.95, 46.29, 125.68) mm, rotated rx -180 ry 0 rz 180 deg; joints [-30.069, 57.069, -88.688, 34.211, 116.982, 17.144]
  Call Extruder(604.07595)
  MoveL 8960 to (240.02, 46.51, 125.68) mm, rotated rx 180 ry 0 rz 180 deg; joints [-30.168, 57.087, -88.687, 34.312, 116.936, 17.179]
  MoveL 8961 to (240.02, 46.51, 125.68) mm, rotated rx 180 ry 0 rz 180 deg; joints [-30.168, 57.087, -88.687, 34.312, 116.936, 17.179]
  Call Extruder(604.19100)
  MoveL 8962 to (240.06, 46.72, 125.68) mm, rotated rx 180 ry 0 rz 180 deg; joints [-30.263, 57.103, -88.686, 34.409, 116.894, 17.215]
  MoveL 8963 to (240.06, 46.72, 125.68) mm, rotated rx 180 ry 0 rz 180 deg; joints [-30.263, 57.103, -88.686, 34.409, 116.894, 17.215]
  Call Extruder(604.30560)
  MoveL 8964 to (240.11, 46.92, 125.68) mm, rotated rx -180 ry 0 rz 180 deg; joints [-30.358, 57.119, -88.685, 34.506, 116.853, 17.25]
  MoveL 8965 to (240.11, 46.92, 125.68) mm, rotated rx -180 ry 0 rz 180 deg; joints [-30.358, 57.119, -88.685, 34.506, 116.853, 17.25]
  Call Extruder(604.41975)
  MoveL 8966 to (240.15, 47.12, 125.68) mm, rotated rx -180 ry 0 rz 180 deg; joints [-30.453, 57.135, -88.684, 34.602, 116.811, 17.285]
  MoveL 8967 to (240.15, 47.12, 125.68) mm, rotated rx -180 ry 0 rz 180 deg; joints [-30.453, 57.135, -88.684, 34.602, 116.811, 17.285]
  Call Extruder(604.53345)
  MoveL 8968 to (240.2, 47.33, 125.68) mm, rotated rx -180 ry 0 rz -180 deg; joints [-30.548, 57.151, -88.683, 34.699, 116.769, 17.32]
  MoveL 8969 to (240.2, 47.33, 125.68) mm, rotated rx -180 ry 0 rz -180 deg; joints [-30.548, 57.151, -88.683, 34.699, 116.769, 17.32]
  Call Extruder(604.65886)
  MoveL 8970 to (240.24, 47.55, 125.68) mm, rotated rx -180 ry 0 rz 180 deg; joints [-30.653, 57.168, -88.682, 34.806, 116.722, 17.359]
  MoveL 8971 to (240.24, 47.55, 125.68) mm, rotated rx -180 ry 0 rz 180 deg; joints [-30.653, 57.168, -88.682, 34.806, 116.722, 17.359]
  Call Extruder(604.79583)
  MoveL 8972 to (240.29, 47.8, 125.68) mm, rotated rx -180 ry 0 rz 180 deg; joints [-30.768, 57.187, -88.68, 34.923, 116.671, 17.401]
  MoveL 8973 to (240.29, 47.8, 125.68) mm, rotated rx -180 ry 0 rz 180 deg; joints [-30.768, 57.187, -88.68, 34.923, 116.671, 17.401]
  Call Extruder(604.93220)
  MoveL 8974 to (240.34, 48.05, 125.68) mm, rotated rx -180 ry 0 rz 180 deg; joints [-30.884, 57.206, -88.679, 35.041, 116.62, 17.444]
  MoveL 8975 to (240.34, 48.05, 125.68) mm, rotated rx -180 ry 0 rz 180 deg; joints [-30.884, 57.206, -88.679, 35.041, 116.62, 17.444]
  Call Extruder(605.06796)
  MoveL 8976 to (240.39, 48.3, 125.68) mm, rotated rx 180 ry 0 rz 180 deg; joints [-30.999, 57.225, -88.678, 35.158, 116.569, 17.486]
  MoveL 8977 to (240.39, 48.3, 125.68) mm, rotated rx 180 ry 0 rz 180 deg; joints [-30.999, 57.225, -88.678, 35.158, 116.569, 17.486]
  Call Extruder(605.20311)
  MoveL 8978 to (240.44, 48.55, 125.68) mm, rotated rx -180 ry 0 rz 180 deg; joints [-31.114, 57.244, -88.677, 35.275, 116.518, 17.528]
  MoveL 8979 to (240.44, 48.55, 125.68) mm, rotated rx -180 ry 0 rz 180 deg; joints [-31.114, 57.244, -88.677, 35.275, 116.518, 17.528]
  Call Extruder(605.33764)
  MoveL 8980 to (240.49, 48.8, 125.68) mm, rotated rx -180 ry 0 rz 180 deg; joints [-31.228, 57.263, -88.675, 35.39, 116.467, 17.569]
  MoveL 8981 to (240.49, 48.8, 125.68) mm, rotated rx -180 ry 0 rz 180 deg; joints [-31.228, 57.263, -88.675, 35.39, 116.467, 17.569]
  Call Extruder(605.47157)
  MoveL 8982 to (240.54, 49.05, 125.68) mm, rotated rx -180 ry 0 rz 180 deg; joints [-31.342, 57.282, -88.674, 35.506, 116.416, 17.61]
  MoveL 8983 to (240.54, 49.05, 125.68) mm, rotated rx -180 ry 0 rz 180 deg; joints [-31.342, 57.282, -88.674, 35.506, 116.416, 17.61]
  Call Extruder(605.61944)
  MoveL 8984 to (240.59, 49.33, 125.68) mm, rotated rx -180 ry 0 rz 180 deg; joints [-31.47, 57.302, -88.673, 35.636, 116.359, 17.656]
  MoveL 8985 to (240.59, 49.33, 125.68) mm, rotated rx -180 ry 0 rz 180 deg; joints [-31.47, 57.302, -88.673, 35.636, 116.359, 17.656]
  Call Extruder(605.78118)
  MoveL 8986 to (240.64, 49.63, 125.68) mm, rotated rx -180 ry 0 rz 180 deg; joints [-31.612, 57.325, -88.671, 35.78, 116.297, 17.707]
  MoveL 8987 to (240.64, 49.63, 125.68) mm, rotated rx -180 ry 0 rz 180 deg; joints [-31.612, 57.325, -88.671, 35.78, 116.297, 17.707]
  Call Extruder(605.94220)
  MoveL 8988 to (240.69, 49.94, 125.68) mm, rotated rx -180 ry 0 rz 180 deg; joints [-31.755, 57.347, -88.67, 35.924, 116.234, 17.759]
  MoveL 8989 to (240.69, 49.94, 125.68) mm, rotated rx -180 ry 0 rz 180 deg; joints [-31.755, 57.347, -88.67, 35.924, 116.234, 17.759]
  Call Extruder(606.10249)
  MoveL 8990 to (240.74, 50.24, 125.68) mm, rotated rx 180 ry 0 rz 180 deg; joints [-31.895, 57.37, -88.668, 36.067, 116.172, 17.809]
  MoveL 8991 to (240.74, 50.24, 125.68) mm, rotated rx 180 ry 0 rz 180 deg; joints [-31.895, 57.37, -88.668, 36.067, 116.172, 17.809]
  Call Extruder(606.26205)
  MoveL 8992 to (240.78, 50.55, 125.68) mm, rotated rx 180 ry 0 rz 180 deg; joints [-32.036, 57.392, -88.667, 36.209, 116.109, 17.859]
  MoveL 8993 to (240.78, 50.55, 125.68) mm, rotated rx 180 ry 0 rz 180 deg; joints [-32.036, 57.392, -88.667, 36.209, 116.109, 17.859]
  Call Extruder(606.42088)
  MoveL 8994 to (240.83, 50.86, 125.68) mm, rotated rx -180 ry 0 rz 180 deg; joints [-32.176, 57.415, -88.665, 36.351, 116.046, 17.908]
  MoveL 8995 to (240.83, 50.86, 125.68) mm, rotated rx -180 ry 0 rz 180 deg; joints [-32.176, 57.415, -88.665, 36.351, 116.046, 17.908]
  Call Extruder(606.59956)
  MoveL 8996 to (240.88, 51.2, 125.68) mm, rotated rx 180 ry 0 rz 180 deg; joints [-32.337, 57.44, -88.663, 36.513, 115.976, 17.965]
  MoveL 8997 to (240.88, 51.2, 125.68) mm, rotated rx 180 ry 0 rz 180 deg; joints [-32.337, 57.44, -88.663, 36.513, 115.976, 17.965]
  Call Extruder(606.79800)
  MoveL 8998 to (240.93, 51.59, 125.68) mm, rotated rx -180 ry 0 rz 180 deg; joints [-32.518, 57.467, -88.661, 36.696, 115.896, 18.029]
  MoveL 8999 to (240.93, 51.59, 125.68) mm, rotated rx -180 ry 0 rz 180 deg; joints [-32.518, 57.467, -88.661, 36.696, 115.896, 18.029]
  Call Extruder(606.99557)
  MoveL 9000 to (240.97, 51.98, 125.68) mm, rotated rx -180 ry 0 rz 180 deg; joints [-32.697, 57.494, -88.659, 36.877, 115.817, 18.092]
  MoveL 9001 to (240.97, 51.98, 125.68) mm, rotated rx -180 ry 0 rz 180 deg; joints [-32.697, 57.494, -88.659, 36.877, 115.817, 18.092]
  Call Extruder(607.19228)
  MoveL 9002 to (241.02, 52.37, 125.68) mm, rotated rx 180 ry 0 rz 180 deg; joints [-32.876, 57.522, -88.657, 37.057, 115.738, 18.155]
  MoveL 9003 to (241.02, 52.37, 125.68) mm, rotated rx 180 ry 0 rz 180 deg; joints [-32.876, 57.522, -88.657, 37.057, 115.738, 18.155]
  Call Extruder(607.38812)
  MoveL 9004 to (241.06, 52.75, 125.68) mm, rotated rx -180 ry 0 rz 180 deg; joints [-33.055, 57.549, -88.655, 37.236, 115.659, 18.217]
  MoveL 9005 to (241.06, 52.75, 125.68) mm, rotated rx -180 ry 0 rz 180 deg; joints [-33.055, 57.549, -88.655, 37.236, 115.659, 18.217]
  Call Extruder(607.68356)
  MoveL 9006 to (241.11, 53.34, 125.68) mm, rotated rx 180 ry 0 rz 180 deg; joints [-33.331, 57.589, -88.652, 37.515, 115.538, 18.314]
  MoveL 9007 to (241.11, 53.34, 125.68) mm, rotated rx 180 ry 0 rz 180 deg; joints [-33.331, 57.589, -88.652, 37.515, 115.538, 18.314]
  Call Extruder(607.97766)
  MoveL 9008 to (241.16, 53.93, 125.68) mm, rotated rx -180 ry 0 rz 180 deg; joints [-33.606, 57.629, -88.649, 37.791, 115.417, 18.408]
  MoveL 9009 to (241.16, 53.93, 125.68) mm, rotated rx -180 ry 0 rz 180 deg; joints [-33.606, 57.629, -88.649, 37.791, 115.417, 18.408]
  Call Extruder(608.27044)
  MoveL 9010 to (241.2, 54.52, 125.68) mm, rotated rx 180 ry 0 rz 180 deg; joints [-33.878, 57.67, -88.646, 38.065, 115.296, 18.501]
  MoveL 9011 to (241.2, 54.52, 125.68) mm, rotated rx 180 ry 0 rz 180 deg; joints [-33.878, 57.67, -88.646, 38.065, 115.296, 18.501]
  Call Extruder(608.84389)
  MoveL 9012 to (241.25, 55.68, 125.68) mm, rotated rx -180 ry 0 rz 180 deg; joints [-34.425, 57.746, -88.639, 38.613, 115.058, 18.688]
  MoveL 9013 to (241.25, 55.68, 125.68) mm, rotated rx -180 ry 0 rz 180 deg; joints [-34.425, 57.746, -88.639, 38.613, 115.058, 18.688]
  Call Extruder(609.55772)
  MoveL 9014 to (241.29, 57.14, 125.68) mm, rotated rx 180 ry 0 rz 180 deg; joints [-35.104, 57.84, -88.632, 39.292, 114.759, 18.916]
  Call Extruder(651.62260)
  MoveL 9015 to (241.29, 142.86, 125.68) mm, rotated rx -180 ry 0 rz 180 deg; joints [-60.361, 64.419, -87.209, 62.32, 101.044, 20.061]
  Call Extruder(652.05103)
  MoveL 9016 to (241.27, 143.74, 125.68) mm, rotated rx 180 ry 0 rz 180 deg; joints [-60.516, 64.488, -87.183, 62.452, 100.947, 20.004]
  MoveL 9017 to (241.27, 143.74, 125.68) mm, rotated rx 180 ry 0 rz 180 deg; joints [-60.516, 64.488, -87.183, 62.452, 100.947, 20.004]
  Call Extruder(652.62448)
  MoveL 9018 to (241.22, 144.9, 125.68) mm, rotated rx 180 ry 0 rz 180 deg; joints [-60.726, 64.579, -87.149, 62.632, 100.817, 19.929]
  MoveL 9019 to (241.22, 144.9, 125.68) mm, rotated rx 180 ry 0 rz 180 deg; joints [-60.726, 64.579, -87.149, 62.632, 100.817, 19.929]
  Call Extruder(653.05882)
  MoveL 9020 to (241.18, 145.77, 125.68) mm, rotated rx -180 ry 0 rz 180 deg; joints [-60.887, 64.647, -87.123, 62.77, 100.719, 19.872]
  MoveL 9021 to (241.18, 145.77, 125.68) mm, rotated rx -180 ry 0 rz 180 deg; joints [-60.887, 64.647, -87.123, 62.77, 100.719, 19.872]
  Call Extruder(653.35293)
  MoveL 9022 to (241.13, 146.36, 125.68) mm, rotated rx -180 ry 0 rz 180 deg; joints [-61, 64.692, -87.105, 62.867, 100.653, 19.836]
  MoveL 9023 to (241.13, 146.36, 125.68) mm, rotated rx -180 ry 0 rz 180 deg; joints [-61, 64.692, -87.105, 62.867, 100.653, 19.836]
  Call Extruder(653.64837)
  MoveL 9024 to (241.09, 146.95, 125.68) mm, rotated rx 180 ry 0 rz 180 deg; joints [-61.111, 64.737, -87.088, 62.964, 100.586, 19.799]
  MoveL 9025 to (241.09, 146.95, 125.68) mm, rotated rx 180 ry 0 rz 180 deg; joints [-61.111, 64.737, -87.088, 62.964, 100.586, 19.799]
  Call Extruder(653.89462)
  MoveL 9026 to (241.04, 147.44, 125.68) mm, rotated rx -180 ry 0 rz 180 deg; joints [-61.205, 64.774, -87.073, 63.045, 100.531, 19.769]
  MoveL 9027 to (241.04, 147.44, 125.68) mm, rotated rx -180 ry 0 rz 180 deg; joints [-61.205, 64.774, -87.073, 63.045, 100.531, 19.769]
  Call Extruder(654.09133)
  MoveL 9028 to (240.99, 147.83, 125.68) mm, rotated rx 180 ry 0 rz 180 deg; joints [-61.282, 64.803, -87.062, 63.112, 100.487, 19.746]
  MoveL 9029 to (240.99, 147.83, 125.68) mm, rotated rx 180 ry 0 rz 180 deg; joints [-61.282, 64.803, -87.062, 63.112, 100.487, 19.746]
  Call Extruder(654.28890)
  MoveL 9030 to (240.95, 148.22, 125.68) mm, rotated rx -180 ry 0 rz 180 deg; joints [-61.359, 64.832, -87.051, 63.179, 100.443, 19.723]
  MoveL 9031 to (240.95, 148.22, 125.68) mm, rotated rx -180 ry 0 rz 180 deg; joints [-61.359, 64.832, -87.051, 63.179, 100.443, 19.723]
  Call Extruder(654.48734)
  MoveL 9032 to (240.9, 148.6, 125.68) mm, rotated rx -180 ry 0 rz 180 deg; joints [-61.436, 64.86, -87.039, 63.246, 100.399, 19.699]
  MoveL 9033 to (240.9, 148.6, 125.68) mm, rotated rx -180 ry 0 rz 180 deg; joints [-61.436, 64.86, -87.039, 63.246, 100.399, 19.699]
  Call Extruder(654.68665)
  MoveL 9034 to (240.86, 148.99, 125.68) mm, rotated rx 180 ry 0 rz 180 deg; joints [-61.512, 64.889, -87.028, 63.312, 100.355, 19.676]
  MoveL 9035 to (240.86, 148.99, 125.68) mm, rotated rx 180 ry 0 rz 180 deg; joints [-61.512, 64.889, -87.028, 63.312, 100.355, 19.676]
  Call Extruder(654.84549)
  MoveL 9036 to (240.81, 149.3, 125.68) mm, rotated rx -180 ry 0 rz 180 deg; joints [-61.575, 64.912, -87.019, 63.368, 100.32, 19.658]
  MoveL 9037 to (240.81, 149.3, 125.68) mm, rotated rx -180 ry 0 rz 180 deg; joints [-61.575, 64.912, -87.019, 63.368, 100.32, 19.658]
  Call Extruder(655.00505)
  MoveL 9038 to (240.76, 149.6, 125.68) mm, rotated rx -180 ry 0 rz 180 deg; joints [-61.639, 64.934, -87.01, 63.424, 100.284, 19.641]
  MoveL 9039 to (240.76, 149.6, 125.68) mm, rotated rx -180 ry 0 rz 180 deg; joints [-61.639, 64.934, -87.01, 63.424, 100.284, 19.641]
  Call Extruder(655.16534)
  MoveL 9040 to (240.71, 149.91, 125.68) mm, rotated rx -180 ry 0 rz 180 deg; joints [-61.702, 64.956, -87.001, 63.479, 100.249, 19.623]
  MoveL 9041 to (240.71, 149.91, 125.68) mm, rotated rx -180 ry 0 rz 180 deg; joints [-61.702, 64.956, -87.001, 63.479, 100.249, 19.623]
  Call Extruder(655.32635)
  MoveL 9042 to (240.66, 150.21, 125.68) mm, rotated rx -180 ry 0 rz 180 deg; joints [-61.765, 64.978, -86.992, 63.534, 100.214, 19.606]
  MoveL 9043 to (240.66, 150.21, 125.68) mm, rotated rx -180 ry 0 rz 180 deg; joints [-61.765, 64.978, -86.992, 63.534, 100.214, 19.606]
  Call Extruder(655.48810)
  MoveL 9044 to (240.61, 150.52, 125.68) mm, rotated rx -180 ry 0 rz -180 deg; joints [-61.828, 65, -86.983, 63.589, 100.179, 19.588]
  MoveL 9045 to (240.61, 150.52, 125.68) mm, rotated rx -180 ry 0 rz -180 deg; joints [-61.828, 65, -86.983, 63.589, 100.179, 19.588]
  Call Extruder(655.65057)
  MoveL 9046 to (240.56, 150.83, 125.68) mm, rotated rx 180 ry 0 rz 180 deg; joints [-61.891, 65.023, -86.974, 63.645, 100.144, 19.57]
  MoveL 9047 to (240.56, 150.83, 125.68) mm, rotated rx 180 ry 0 rz 180 deg; joints [-61.891, 65.023, -86.974, 63.645, 100.144, 19.57]
  Call Extruder(655.78449)
  MoveL 9048 to (240.52, 151.08, 125.68) mm, rotated rx -180 ry 0 rz -180 deg; joints [-61.944, 65.04, -86.966, 63.692, 100.115, 19.556]
  MoveL 9049 to (240.52, 151.08, 125.68) mm, rotated rx -180 ry 0 rz -180 deg; joints [-61.944, 65.04, -86.966, 63.692, 100.115, 19.556]
  Call Extruder(655.91903)
  MoveL 9050 to (240.47, 151.32, 125.68) mm, rotated rx -180 ry 0 rz 180 deg; joints [-61.998, 65.058, -86.959, 63.74, 100.086, 19.543]
  MoveL 9051 to (240.47, 151.32, 125.68) mm, rotated rx -180 ry 0 rz 180 deg; joints [-61.998, 65.058, -86.959, 63.74, 100.086, 19.543]
  Call Extruder(656.05418)
  MoveL 9052 to (240.42, 151.57, 125.68) mm, rotated rx 180 ry 0 rz 180 deg; joints [-62.052, 65.076, -86.952, 63.787, 100.057, 19.529]
  MoveL 9053 to (240.42, 151.57, 125.68) mm, rotated rx 180 ry 0 rz 180 deg; joints [-62.052, 65.076, -86.952, 63.787, 100.057, 19.529]
  Call Extruder(656.18994)
  MoveL 9054 to (240.37, 151.82, 125.68) mm, rotated rx -180 ry 0 rz 180 deg; joints [-62.105, 65.093, -86.944, 63.834, 100.028, 19.515]
  MoveL 9055 to (240.37, 151.82, 125.68) mm, rotated rx -180 ry 0 rz 180 deg; joints [-62.105, 65.093, -86.944, 63.834, 100.028, 19.515]
  Call Extruder(656.32630)
  MoveL 9056 to (240.32, 152.07, 125.68) mm, rotated rx -180 ry 0 rz 180 deg; joints [-62.159, 65.111, -86.937, 63.882, 99.999, 19.501]
  MoveL 9057 to (240.32, 152.07, 125.68) mm, rotated rx -180 ry 0 rz 180 deg; joints [-62.159, 65.111, -86.937, 63.882, 99.999, 19.501]
  Call Extruder(656.46328)
  MoveL 9058 to (240.27, 152.32, 125.68) mm, rotated rx -180 ry 0 rz 180 deg; joints [-62.212, 65.129, -86.93, 63.928, 99.97, 19.487]
  MoveL 9059 to (240.27, 152.32, 125.68) mm, rotated rx -180 ry 0 rz 180 deg; joints [-62.212, 65.129, -86.93, 63.928, 99.97, 19.487]
  Call Extruder(656.60087)
  MoveL 9060 to (240.22, 152.57, 125.68) mm, rotated rx 180 ry 0 rz 180 deg; joints [-62.265, 65.147, -86.922, 63.975, 99.942, 19.473]
  MoveL 9061 to (240.22, 152.57, 125.68) mm, rotated rx 180 ry 0 rz 180 deg; joints [-62.265, 65.147, -86.922, 63.975, 99.942, 19.473]
  Call Extruder(656.71457)
  MoveL 9062 to (240.17, 152.77, 125.68) mm, rotated rx -180 ry 0 rz -180 deg; joints [-62.31, 65.161, -86.916, 64.015, 99.918, 19.462]
  MoveL 9063 to (240.17, 152.77, 125.68) mm, rotated rx -180 ry 0 rz -180 deg; joints [-62.31, 65.161, -86.916, 64.015, 99.918, 19.462]
  Call Extruder(656.82872)
  MoveL 9064 to (240.13, 152.98, 125.68) mm, rotated rx 180 ry 0 rz 180 deg; joints [-62.355, 65.175, -86.91, 64.055, 99.894, 19.451]
  MoveL 9065 to (240.13, 152.98, 125.68) mm, rotated rx 180 ry 0 rz 180 deg; joints [-62.355, 65.175, -86.91, 64.055, 99.894, 19.451]
  Call Extruder(656.94332)
  MoveL 9066 to (240.08, 153.18, 125.68) mm, rotated rx -180 ry 0 rz 180 deg; joints [-62.399, 65.19, -86.904, 64.094, 99.87, 19.439]
  MoveL 9067 to (240.08, 153.18, 125.68) mm, rotated rx -180 ry 0 rz 180 deg; joints [-62.399, 65.19, -86.904, 64.094, 99.87, 19.439]
  Call Extruder(657.05837)
  MoveL 9068 to (240.04, 153.39, 125.68) mm, rotated rx 180 ry 0 rz 180 deg; joints [-62.444, 65.204, -86.898, 64.133, 99.847, 19.428]
  MoveL 9069 to (240.04, 153.39, 125.68) mm, rotated rx 180 ry 0 rz 180 deg; joints [-62.444, 65.204, -86.898, 64.133, 99.847, 19.428]
  Call Extruder(657.18060)
  MoveL 9070 to (239.98, 153.6, 125.68) mm, rotated rx -180 ry 0 rz 180 deg; joints [-62.493, 65.219, -86.892, 64.177, 99.821, 19.417]
  MoveL 9071 to (239.98, 153.6, 125.68) mm, rotated rx -180 ry 0 rz 180 deg; joints [-62.493, 65.219, -86.892, 64.177, 99.821, 19.417]
  Call Extruder(657.31026)
  MoveL 9072 to (239.92, 153.82, 125.68) mm, rotated rx 180 ry 0 rz -180 deg; joints [-62.547, 65.234, -86.886, 64.225, 99.794, 19.406]
  MoveL 9073 to (239.92, 153.82, 125.68) mm, rotated rx 180 ry 0 rz -180 deg; joints [-62.547, 65.234, -86.886, 64.225, 99.794, 19.406]
  Call Extruder(657.44048)
  MoveL 9074 to (239.85, 154.05, 125.68) mm, rotated rx -180 ry 0 rz 180 deg; joints [-62.601, 65.249, -86.88, 64.274, 99.767, 19.396]
  MoveL 9075 to (239.85, 154.05, 125.68) mm, rotated rx -180 ry 0 rz 180 deg; joints [-62.601, 65.249, -86.88, 64.274, 99.767, 19.396]
  Call Extruder(657.57127)
  MoveL 9076 to (239.78, 154.27, 125.68) mm, rotated rx -180 ry 0 rz 180 deg; joints [-62.654, 65.264, -86.873, 64.322, 99.74, 19.385]
  MoveL 9077 to (239.78, 154.27, 125.68) mm, rotated rx -180 ry 0 rz 180 deg; joints [-62.654, 65.264, -86.873, 64.322, 99.74, 19.385]
  Call Extruder(657.70262)
  MoveL 9078 to (239.71, 154.5, 125.68) mm, rotated rx -180 ry 0 rz 180 deg; joints [-62.708, 65.279, -86.867, 64.37, 99.713, 19.374]
  MoveL 9079 to (239.71, 154.5, 125.68) mm, rotated rx -180 ry 0 rz 180 deg; joints [-62.708, 65.279, -86.867, 64.37, 99.713, 19.374]
  Call Extruder(657.81453)
  MoveL 9080 to (239.65, 154.68, 125.68) mm, rotated rx 180 ry 0 rz 180 deg; joints [-62.754, 65.291, -86.862, 64.411, 99.69, 19.365]
  MoveL 9081 to (239.65, 154.68, 125.68) mm, rotated rx 180 ry 0 rz 180 deg; joints [-62.754, 65.291, -86.862, 64.411, 99.69, 19.365]
  Call Extruder(657.92687)
  MoveL 9082 to (239.59, 154.87, 125.68) mm, rotated rx -180 ry 0 rz 180 deg; joints [-62.801, 65.303, -86.856, 64.453, 99.667, 19.356]
  MoveL 9083 to (239.59, 154.87, 125.68) mm, rotated rx -180 ry 0 rz 180 deg; joints [-62.801, 65.303, -86.856, 64.453, 99.667, 19.356]
  Call Extruder(658.03966)
  MoveL 9084 to (239.53, 155.06, 125.68) mm, rotated rx 180 ry 0 rz -180 deg; joints [-62.847, 65.316, -86.851, 64.495, 99.644, 19.348]
  MoveL 9085 to (239.53, 155.06, 125.68) mm, rotated rx 180 ry 0 rz -180 deg; joints [-62.847, 65.316, -86.851, 64.495, 99.644, 19.348]
  Call Extruder(658.15290)
  MoveL 9086 to (239.47, 155.25, 125.68) mm, rotated rx 180 ry 0 rz -180 deg; joints [-62.893, 65.328, -86.846, 64.536, 99.621, 19.339]
  MoveL 9087 to (239.47, 155.25, 125.68) mm, rotated rx 180 ry 0 rz -180 deg; joints [-62.893, 65.328, -86.846, 64.536, 99.621, 19.339]
  Call Extruder(658.26658)
  MoveL 9088 to (239.41, 155.44, 125.68) mm, rotated rx 180 ry 0 rz 180 deg; joints [-62.939, 65.341, -86.84, 64.577, 99.598, 19.33]
  MoveL 9089 to (239.41, 155.44, 125.68) mm, rotated rx 180 ry 0 rz 180 deg; joints [-62.939, 65.341, -86.84, 64.577, 99.598, 19.33]
  Call Extruder(658.44854)
  MoveL 9090 to (239.29, 155.73, 125.68) mm, rotated rx -180 ry 0 rz -180 deg; joints [-63.018, 65.359, -86.833, 64.649, 99.561, 19.319]
  MoveL 9091 to (239.29, 155.73, 125.68) mm, rotated rx -180 ry 0 rz -180 deg; joints [-63.018, 65.359, -86.833, 64.649, 99.561, 19.319]
  Call Extruder(658.63125)
  MoveL 9092 to (239.17, 156.02, 125.68) mm, rotated rx 180 ry 0 rz -180 deg; joints [-63.097, 65.377, -86.825, 64.72, 99.523, 19.307]
  MoveL 9093 to (239.17, 156.02, 125.68) mm, rotated rx 180 ry 0 rz -180 deg; joints [-63.097, 65.377, -86.825, 64.72, 99.523, 19.307]
  Call Extruder(658.80168)
  MoveL 9094 to (239.05, 156.29, 125.68) mm, rotated rx 180 ry 0 rz 180 deg; joints [-63.17, 65.394, -86.817, 64.787, 99.489, 19.297]
  MoveL 9095 to (239.05, 156.29, 125.68) mm, rotated rx 180 ry 0 rz 180 deg; joints [-63.17, 65.394, -86.817, 64.787, 99.489, 19.297]
  Call Extruder(658.95972)
  MoveL 9096 to (238.94, 156.54, 125.68) mm, rotated rx 180 ry 0 rz -180 deg; joints [-63.238, 65.41, -86.811, 64.849, 99.457, 19.287]
  MoveL 9097 to (238.94, 156.54, 125.68) mm, rotated rx 180 ry 0 rz -180 deg; joints [-63.238, 65.41, -86.811, 64.849, 99.457, 19.287]
  Call Extruder(659.11835)
  MoveL 9098 to (238.84, 156.79, 125.68) mm, rotated rx -180 ry 0 rz 180 deg; joints [-63.306, 65.425, -86.804, 64.91, 99.425, 19.277]
  MoveL 9099 to (238.84, 156.79, 125.68) mm, rotated rx -180 ry 0 rz 180 deg; joints [-63.306, 65.425, -86.804, 64.91, 99.425, 19.277]
  Call Extruder(659.32451)
  MoveL 9100 to (238.66, 157.09, 125.68) mm, rotated rx -180 ry 0 rz 180 deg; joints [-63.401, 65.442, -86.797, 64.998, 99.383, 19.269]
  MoveL 9101 to (238.66, 157.09, 125.68) mm, rotated rx -180 ry 0 rz 180 deg; joints [-63.401, 65.442, -86.797, 64.998, 99.383, 19.269]
  Call Extruder(659.53144)
  MoveL 9102 to (238.49, 157.4, 125.68) mm, rotated rx -180 ry 0 rz -180 deg; joints [-63.497, 65.459, -86.789, 65.086, 99.341, 19.262]
  MoveL 9103 to (238.49, 157.4, 125.68) mm, rotated rx -180 ry 0 rz -180 deg; joints [-63.497, 65.459, -86.789, 65.086, 99.341, 19.262]
  Call Extruder(659.73916)
  MoveL 9104 to (238.31, 157.7, 125.68) mm, rotated rx 180 ry 0 rz 180 deg; joints [-63.592, 65.477, -86.782, 65.173, 99.299, 19.254]
  MoveL 9105 to (238.31, 157.7, 125.68) mm, rotated rx 180 ry 0 rz 180 deg; joints [-63.592, 65.477, -86.782, 65.173, 99.299, 19.254]
  Call Extruder(659.94765)
  MoveL 9106 to (238.13, 158.01, 125.68) mm, rotated rx -180 ry 0 rz 180 deg; joints [-63.687, 65.494, -86.774, 65.26, 99.258, 19.246]
  MoveL 9107 to (238.13, 158.01, 125.68) mm, rotated rx -180 ry 0 rz 180 deg; joints [-63.687, 65.494, -86.774, 65.26, 99.258, 19.246]
  Call Extruder(660.12717)
  MoveL 9108 to (237.96, 158.25, 125.68) mm, rotated rx 180 ry 0 rz 180 deg; joints [-63.774, 65.506, -86.769, 65.34, 99.222, 19.242]
  MoveL 9109 to (237.96, 158.25, 125.68) mm, rotated rx 180 ry 0 rz 180 deg; joints [-63.774, 65.506, -86.769, 65.34, 99.222, 19.242]
  Call Extruder(660.46059)
  MoveL 9110 to (237.63, 158.7, 125.68) mm, rotated rx -180 ry 0 rz 180 deg; joints [-63.934, 65.529, -86.758, 65.489, 99.155, 19.236]
  MoveL 9111 to (237.63, 158.7, 125.68) mm, rotated rx -180 ry 0 rz 180 deg; joints [-63.934, 65.529, -86.758, 65.489, 99.155, 19.236]
  Call Extruder(660.79519)
  MoveL 9112 to (237.3, 159.15, 125.68) mm, rotated rx 180 ry 0 rz 180 deg; joints [-64.094, 65.553, -86.748, 65.636, 99.089, 19.23]
  Call Extruder(661.62314)
  MoveL 9113 to (236.39, 160.19, 125.68) mm, rotated rx -180 ry 0 rz 180 deg; joints [-64.505, 65.6, -86.727, 66.019, 98.925, 19.228]
  Call Extruder(662.45109)
  MoveL 9114 to (235.35, 161.1, 125.68) mm, rotated rx -180 ry 0 rz -180 deg; joints [-64.933, 65.634, -86.712, 66.422, 98.765, 19.246]
  Call Extruder(662.61839)
  MoveL 9115 to (235.13, 161.27, 125.68) mm, rotated rx 180 ry 0 rz 180 deg; joints [-65.021, 65.638, -86.71, 66.505, 98.733, 19.252]
  MoveL 9116 to (235.13, 161.27, 125.68) mm, rotated rx 180 ry 0 rz 180 deg; joints [-65.021, 65.638, -86.71, 66.505, 98.733, 19.252]
  Call Extruder(662.95182)
  MoveL 9117 to (234.68, 161.59, 125.68) mm, rotated rx -180 ry 0 rz 180 deg; joints [-65.197, 65.648, -86.706, 66.671, 98.669, 19.265]
  MoveL 9118 to (234.68, 161.59, 125.68) mm, rotated rx -180 ry 0 rz 180 deg; joints [-65.197, 65.648, -86.706, 66.671, 98.669, 19.265]
  Call Extruder(663.28405)
  MoveL 9119 to (234.22, 161.92, 125.68) mm, rotated rx -180 ry 0 rz -180 deg; joints [-65.374, 65.658, -86.701, 66.838, 98.605, 19.277]
  MoveL 9120 to (234.22, 161.92, 125.68) mm, rotated rx -180 ry 0 rz -180 deg; joints [-65.374, 65.658, -86.701, 66.838, 98.605, 19.277]
  Call Extruder(663.40172)
  MoveL 9121 to (234.05, 162.02, 125.68) mm, rotated rx 180 ry 0 rz 180 deg; joints [-65.437, 65.659, -86.701, 66.898, 98.584, 19.284]
  MoveL 9122 to (234.05, 162.02, 125.68) mm, rotated rx 180 ry 0 rz 180 deg; joints [-65.437, 65.659, -86.701, 66.898, 98.584, 19.284]
  Call Extruder(663.60945)
  MoveL 9123 to (233.75, 162.2, 125.68) mm, rotated rx -180 ry 0 rz 180 deg; joints [-65.549, 65.662, -86.699, 67.004, 98.545, 19.296]
  MoveL 9124 to (233.75, 162.2, 125.68) mm, rotated rx -180 ry 0 rz 180 deg; joints [-65.549, 65.662, -86.699, 67.004, 98.545, 19.296]
  Call Extruder(663.81640)
  MoveL 9125 to (233.45, 162.37, 125.68) mm, rotated rx -180 ry 0 rz 180 deg; joints [-65.662, 65.665, -86.698, 67.111, 98.506, 19.308]
  MoveL 9126 to (233.45, 162.37, 125.68) mm, rotated rx -180 ry 0 rz 180 deg; joints [-65.662, 65.665, -86.698, 67.111, 98.506, 19.308]
  Call Extruder(664.02257)
  MoveL 9127 to (233.14, 162.55, 125.68) mm, rotated rx -180 ry 0 rz 180 deg; joints [-65.774, 65.668, -86.697, 67.217, 98.467, 19.319]
  MoveL 9128 to (233.14, 162.55, 125.68) mm, rotated rx -180 ry 0 rz 180 deg; joints [-65.774, 65.668, -86.697, 67.217, 98.467, 19.319]
  Call Extruder(664.20424)
  MoveL 9129 to (232.87, 162.69, 125.68) mm, rotated rx 180 ry 0 rz 180 deg; joints [-65.874, 65.67, -86.696, 67.313, 98.433, 19.331]
  MoveL 9130 to (232.87, 162.69, 125.68) mm, rotated rx 180 ry 0 rz 180 deg; joints [-65.874, 65.67, -86.696, 67.313, 98.433, 19.331]
  Call Extruder(664.36221)
  MoveL 9131 to (232.62, 162.8, 125.68) mm, rotated rx -180 ry 0 rz 180 deg; joints [-65.961, 65.669, -86.696, 67.396, 98.405, 19.344]
  MoveL 9132 to (232.62, 162.8, 125.68) mm, rotated rx -180 ry 0 rz 180 deg; joints [-65.961, 65.669, -86.696, 67.396, 98.405, 19.344]
  Call Extruder(664.51957)
  MoveL 9133 to (232.37, 162.91, 125.68) mm, rotated rx 180 ry 0 rz 180 deg; joints [-66.048, 65.669, -86.696, 67.479, 98.376, 19.357]
  MoveL 9134 to (232.37, 162.91, 125.68) mm, rotated rx 180 ry 0 rz 180 deg; joints [-66.048, 65.669, -86.696, 67.479, 98.376, 19.357]
  Call Extruder(664.70231)
  MoveL 9135 to (232.07, 163.03, 125.68) mm, rotated rx 180 ry 0 rz -180 deg; joints [-66.149, 65.668, -86.697, 67.576, 98.343, 19.372]
  MoveL 9136 to (232.07, 163.03, 125.68) mm, rotated rx 180 ry 0 rz -180 deg; joints [-66.149, 65.668, -86.697, 67.576, 98.343, 19.372]
  Call Extruder(664.88429)
  MoveL 9137 to (231.78, 163.15, 125.68) mm, rotated rx 180 ry 0 rz 180 deg; joints [-66.251, 65.668, -86.697, 67.673, 98.309, 19.387]
  MoveL 9138 to (231.78, 163.15, 125.68) mm, rotated rx 180 ry 0 rz 180 deg; joints [-66.251, 65.668, -86.697, 67.673, 98.309, 19.387]
  Call Extruder(665.03163)
  MoveL 9139 to (231.54, 163.24, 125.68) mm, rotated rx 180 ry 0 rz 180 deg; joints [-66.333, 65.666, -86.697, 67.751, 98.283, 19.4]
  MoveL 9140 to (231.54, 163.24, 125.68) mm, rotated rx 180 ry 0 rz 180 deg; joints [-66.333, 65.666, -86.697, 67.751, 98.283, 19.4]
  Call Extruder(665.14485)
  MoveL 9141 to (231.35, 163.3, 125.68) mm, rotated rx 180 ry 0 rz 180 deg; joints [-66.397, 65.665, -86.698, 67.812, 98.262, 19.41]
  MoveL 9142 to (231.35, 163.3, 125.68) mm, rotated rx 180 ry 0 rz 180 deg; joints [-66.397, 65.665, -86.698, 67.812, 98.262, 19.41]
  Call Extruder(665.25763)
  MoveL 9143 to (231.17, 163.36, 125.68) mm, rotated rx 180 ry 0 rz 180 deg; joints [-66.46, 65.663, -86.699, 67.873, 98.242, 19.421]
  MoveL 9144 to (231.17, 163.36, 125.68) mm, rotated rx 180 ry 0 rz 180 deg; joints [-66.46, 65.663, -86.699, 67.873, 98.242, 19.421]
  Call Extruder(665.36996)
  MoveL 9145 to (230.98, 163.42, 125.68) mm, rotated rx -180 ry 0 rz -180 deg; joints [-66.524, 65.661, -86.7, 67.934, 98.222, 19.432]
  MoveL 9146 to (230.98, 163.42, 125.68) mm, rotated rx -180 ry 0 rz -180 deg; joints [-66.524, 65.661, -86.7, 67.934, 98.222, 19.432]
  Call Extruder(665.48185)
  MoveL 9147 to (230.79, 163.48, 125.68) mm, rotated rx -180 ry 0 rz 180 deg; joints [-66.587, 65.66, -86.7, 67.995, 98.202, 19.443]
  MoveL 9148 to (230.79, 163.48, 125.68) mm, rotated rx -180 ry 0 rz 180 deg; joints [-66.587, 65.66, -86.7, 67.995, 98.202, 19.443]
  Call Extruder(665.60326)
  MoveL 9149 to (230.58, 163.55, 125.68) mm, rotated rx -180 ry 0 rz 180 deg; joints [-66.656, 65.658, -86.701, 68.061, 98.18, 19.455]
  MoveL 9150 to (230.58, 163.55, 125.68) mm, rotated rx -180 ry 0 rz 180 deg; joints [-66.656, 65.658, -86.701, 68.061, 98.18, 19.455]
  Call Extruder(665.73407)
  MoveL 9151 to (230.36, 163.62, 125.68) mm, rotated rx -180 ry 0 rz 180 deg; joints [-66.731, 65.655, -86.702, 68.132, 98.156, 19.469]
  MoveL 9152 to (230.36, 163.62, 125.68) mm, rotated rx -180 ry 0 rz 180 deg; joints [-66.731, 65.655, -86.702, 68.132, 98.156, 19.469]
  Call Extruder(665.86432)
  MoveL 9153 to (230.14, 163.68, 125.68) mm, rotated rx -180 ry 0 rz -180 deg; joints [-66.805, 65.653, -86.703, 68.204, 98.133, 19.482]
  MoveL 9154 to (230.14, 163.68, 125.68) mm, rotated rx -180 ry 0 rz -180 deg; joints [-66.805, 65.653, -86.703, 68.204, 98.133, 19.482]
  Call Extruder(665.99400)
  MoveL 9155 to (229.91, 163.75, 125.68) mm, rotated rx 180 ry 0 rz 180 deg; joints [-66.88, 65.651, -86.704, 68.276, 98.109, 19.495]
  MoveL 9156 to (229.91, 163.75, 125.68) mm, rotated rx 180 ry 0 rz 180 deg; joints [-66.88, 65.651, -86.704, 68.276, 98.109, 19.495]
  Call Extruder(666.12312)
  MoveL 9157 to (229.69, 163.82, 125.68) mm, rotated rx -180 ry 0 rz 180 deg; joints [-66.955, 65.649, -86.705, 68.347, 98.085, 19.508]
  MoveL 9158 to (229.69, 163.82, 125.68) mm, rotated rx -180 ry 0 rz 180 deg; joints [-66.955, 65.649, -86.705, 68.347, 98.085, 19.508]
  Call Extruder(666.23819)
  MoveL 9159 to (229.48, 163.86, 125.68) mm, rotated rx 180 ry 0 rz 180 deg; joints [-67.021, 65.645, -86.707, 68.411, 98.065, 19.521]
  MoveL 9160 to (229.48, 163.86, 125.68) mm, rotated rx 180 ry 0 rz 180 deg; joints [-67.021, 65.645, -86.707, 68.411, 98.065, 19.521]
  Call Extruder(666.35282)
  MoveL 9161 to (229.28, 163.91, 125.68) mm, rotated rx -180 ry 0 rz 180 deg; joints [-67.087, 65.642, -86.708, 68.474, 98.045, 19.535]
  MoveL 9162 to (229.28, 163.91, 125.68) mm, rotated rx -180 ry 0 rz 180 deg; joints [-67.087, 65.642, -86.708, 68.474, 98.045, 19.535]
  Call Extruder(666.46699)
  MoveL 9163 to (229.08, 163.95, 125.68) mm, rotated rx -180 ry 0 rz 180 deg; joints [-67.153, 65.638, -86.71, 68.538, 98.024, 19.548]
  MoveL 9164 to (229.08, 163.95, 125.68) mm, rotated rx -180 ry 0 rz 180 deg; joints [-67.153, 65.638, -86.71, 68.538, 98.024, 19.548]
  Call Extruder(666.58070)
  MoveL 9165 to (228.87, 164, 125.68) mm, rotated rx -180 ry 0 rz -180 deg; joints [-67.22, 65.635, -86.711, 68.602, 98.004, 19.562]
  MoveL 9166 to (228.87, 164, 125.68) mm, rotated rx -180 ry 0 rz -180 deg; joints [-67.22, 65.635, -86.711, 68.602, 98.004, 19.562]
  Call Extruder(666.70613)
  MoveL 9167 to (228.64, 164.04, 125.68) mm, rotated rx -180 ry 0 rz -180 deg; joints [-67.293, 65.631, -86.713, 68.672, 97.981, 19.577]
  MoveL 9168 to (228.64, 164.04, 125.68) mm, rotated rx -180 ry 0 rz -180 deg; joints [-67.293, 65.631, -86.713, 68.672, 97.981, 19.577]
  Call Extruder(666.84310)
  MoveL 9169 to (228.4, 164.09, 125.68) mm, rotated rx 180 ry 0 rz 180 deg; joints [-67.373, 65.627, -86.715, 68.749, 97.957, 19.593]
  MoveL 9170 to (228.4, 164.09, 125.68) mm, rotated rx 180 ry 0 rz 180 deg; joints [-67.373, 65.627, -86.715, 68.749, 97.957, 19.593]
  Call Extruder(666.97947)
  MoveL 9171 to (228.15, 164.14, 125.68) mm, rotated rx 180 ry 0 rz 180 deg; joints [-67.453, 65.622, -86.717, 68.826, 97.932, 19.61]
  MoveL 9172 to (228.15, 164.14, 125.68) mm, rotated rx 180 ry 0 rz 180 deg; joints [-67.453, 65.622, -86.717, 68.826, 97.932, 19.61]
  Call Extruder(667.11523)
  MoveL 9173 to (227.9, 164.19, 125.68) mm, rotated rx -180 ry 0 rz 180 deg; joints [-67.534, 65.618, -86.719, 68.904, 97.908, 19.626]
  MoveL 9174 to (227.9, 164.19, 125.68) mm, rotated rx -180 ry 0 rz 180 deg; joints [-67.534, 65.618, -86.719, 68.904, 97.908, 19.626]
  Call Extruder(667.25038)
  MoveL 9175 to (227.65, 164.24, 125.68) mm, rotated rx 180 ry 0 rz 180 deg; joints [-67.614, 65.614, -86.721, 68.981, 97.883, 19.643]
  MoveL 9176 to (227.65, 164.24, 125.68) mm, rotated rx 180 ry 0 rz 180 deg; joints [-67.614, 65.614, -86.721, 68.981, 97.883, 19.643]
  Call Extruder(667.38491)
  MoveL 9177 to (227.4, 164.29, 125.68) mm, rotated rx -180 ry 0 rz 180 deg; joints [-67.695, 65.609, -86.723, 69.058, 97.858, 19.659]
  MoveL 9178 to (227.4, 164.29, 125.68) mm, rotated rx -180 ry 0 rz 180 deg; joints [-67.695, 65.609, -86.723, 69.058, 97.858, 19.659]
  Call Extruder(667.51884)
  MoveL 9179 to (227.15, 164.34, 125.68) mm, rotated rx 180 ry 0 rz -180 deg; joints [-67.775, 65.605, -86.725, 69.135, 97.833, 19.675]
  MoveL 9180 to (227.15, 164.34, 125.68) mm, rotated rx 180 ry 0 rz -180 deg; joints [-67.775, 65.605, -86.725, 69.135, 97.833, 19.675]
  Call Extruder(667.66670)
  MoveL 9181 to (226.87, 164.39, 125.68) mm, rotated rx 180 ry 0 rz -180 deg; joints [-67.864, 65.6, -86.727, 69.221, 97.806, 19.694]
  MoveL 9182 to (226.87, 164.39, 125.68) mm, rotated rx 180 ry 0 rz -180 deg; joints [-67.864, 65.6, -86.727, 69.221, 97.806, 19.694]
  Call Extruder(667.82844)
  MoveL 9183 to (226.57, 164.44, 125.68) mm, rotated rx 180 ry 0 rz -180 deg; joints [-67.961, 65.594, -86.73, 69.314, 97.776, 19.715]
  MoveL 9184 to (226.57, 164.44, 125.68) mm, rotated rx 180 ry 0 rz -180 deg; joints [-67.961, 65.594, -86.73, 69.314, 97.776, 19.715]
  Call Extruder(667.98945)
  MoveL 9185 to (226.26, 164.49, 125.68) mm, rotated rx 180 ry 0 rz -180 deg; joints [-68.059, 65.588, -86.733, 69.408, 97.746, 19.736]
  MoveL 9186 to (226.26, 164.49, 125.68) mm, rotated rx 180 ry 0 rz -180 deg; joints [-68.059, 65.588, -86.733, 69.408, 97.746, 19.736]
  Call Extruder(668.14974)
  MoveL 9187 to (225.95, 164.54, 125.68) mm, rotated rx 180 ry 0 rz -180 deg; joints [-68.156, 65.582, -86.735, 69.502, 97.717, 19.757]
  MoveL 9188 to (225.95, 164.54, 125.68) mm, rotated rx 180 ry 0 rz -180 deg; joints [-68.156, 65.582, -86.735, 69.502, 97.717, 19.757]
  Call Extruder(668.30929)
  MoveL 9189 to (225.65, 164.58, 125.68) mm, rotated rx -180 ry 0 rz 180 deg; joints [-68.254, 65.575, -86.738, 69.596, 97.687, 19.777]
  MoveL 9190 to (225.65, 164.58, 125.68) mm, rotated rx -180 ry 0 rz 180 deg; joints [-68.254, 65.575, -86.738, 69.596, 97.687, 19.777]
  Call Extruder(668.46812)
  MoveL 9191 to (225.34, 164.63, 125.68) mm, rotated rx -180 ry 0 rz 180 deg; joints [-68.351, 65.569, -86.741, 69.689, 97.657, 19.798]
  MoveL 9192 to (225.34, 164.63, 125.68) mm, rotated rx -180 ry 0 rz 180 deg; joints [-68.351, 65.569, -86.741, 69.689, 97.657, 19.798]
  Call Extruder(668.64679)
  MoveL 9193 to (225, 164.68, 125.68) mm, rotated rx 180 ry 0 rz 180 deg; joints [-68.461, 65.562, -86.744, 69.795, 97.623, 19.822]
  MoveL 9194 to (225, 164.68, 125.68) mm, rotated rx 180 ry 0 rz 180 deg; joints [-68.461, 65.562, -86.744, 69.795, 97.623, 19.822]
  Call Extruder(668.84523)
  MoveL 9195 to (224.61, 164.73, 125.68) mm, rotated rx 180 ry 0 rz 180 deg; joints [-68.583, 65.553, -86.748, 69.913, 97.586, 19.849]
  MoveL 9196 to (224.61, 164.73, 125.68) mm, rotated rx 180 ry 0 rz 180 deg; joints [-68.583, 65.553, -86.748, 69.913, 97.586, 19.849]
  Call Extruder(669.04281)
  MoveL 9197 to (224.22, 164.77, 125.68) mm, rotated rx -180 ry 0 rz -180 deg; joints [-68.706, 65.545, -86.752, 70.03, 97.549, 19.876]
  MoveL 9198 to (224.22, 164.77, 125.68) mm, rotated rx -180 ry 0 rz -180 deg; joints [-68.706, 65.545, -86.752, 70.03, 97.549, 19.876]
  Call Extruder(669.23952)
  MoveL 9199 to (223.84, 164.82, 125.68) mm, rotated rx 180 ry 0 rz 180 deg; joints [-68.828, 65.536, -86.755, 70.148, 97.511, 19.903]
  MoveL 9200 to (223.84, 164.82, 125.68) mm, rotated rx 180 ry 0 rz 180 deg; joints [-68.828, 65.536, -86.755, 70.148, 97.511, 19.903]
  Call Extruder(669.43535)
  MoveL 9201 to (223.45, 164.86, 125.68) mm, rotated rx -180 ry 0 rz -180 deg; joints [-68.951, 65.527, -86.759, 70.266, 97.474, 19.93]
  MoveL 9202 to (223.45, 164.86, 125.68) mm, rotated rx -180 ry 0 rz -180 deg; joints [-68.951, 65.527, -86.759, 70.266, 97.474, 19.93]
  Call Extruder(669.73071)
  MoveL 9203 to (222.86, 164.91, 125.68) mm, rotated rx 180 ry 0 rz 180 deg; joints [-69.135, 65.513, -86.766, 70.443, 97.418, 19.973]
  MoveL 9204 to (222.86, 164.91, 125.68) mm, rotated rx 180 ry 0 rz 180 deg; joints [-69.135, 65.513, -86.766, 70.443, 97.418, 19.973]
  Call Extruder(670.02474)
  MoveL 9205 to (222.27, 164.96, 125.68) mm, rotated rx 180 ry 0 rz -180 deg; joints [-69.319, 65.498, -86.772, 70.62, 97.362, 20.015]
  MoveL 9206 to (222.27, 164.96, 125.68) mm, rotated rx 180 ry 0 rz -180 deg; joints [-69.319, 65.498, -86.772, 70.62, 97.362, 20.015]
  Call Extruder(670.31744)
  MoveL 9207 to (221.68, 165, 125.68) mm, rotated rx -180 ry 0 rz -180 deg; joints [-69.504, 65.484, -86.779, 70.797, 97.306, 20.058]
  MoveL 9208 to (221.68, 165, 125.68) mm, rotated rx -180 ry 0 rz -180 deg; joints [-69.504, 65.484, -86.779, 70.797, 97.306, 20.058]
  Call Extruder(670.89088)
  MoveL 9209 to (220.52, 165.05, 125.68) mm, rotated rx -180 ry 0 rz 180 deg; joints [-69.864, 65.452, -86.792, 71.144, 97.197, 20.144]
  MoveL 9210 to (220.52, 165.05, 125.68) mm, rotated rx -180 ry 0 rz 180 deg; joints [-69.864, 65.452, -86.792, 71.144, 97.197, 20.144]
  Call Extruder(671.60489)
  MoveL 9211 to (219.06, 165.09, 125.68) mm, rotated rx -180 ry 0 rz -180 deg; joints [-70.315, 65.411, -86.81, 71.577, 97.06, 20.253]
  Call Extruder(788.45163)
  MoveL 9212 to (-19.06, 165.09, 125.68) mm, rotated rx 180 ry 0 rz 180 deg; joints [-137.325, 70.735, -83.309, 136.632, 80.79, 8.597]
  Call Extruder(788.88023)
  MoveL 9213 to (-19.94, 165.07, 125.68) mm, rotated rx 180 ry 0 rz -180 deg; joints [-137.467, 70.777, -83.268, 136.783, 80.829, 8.517]
  MoveL 9214 to (-19.94, 165.07, 125.68) mm, rotated rx 180 ry 0 rz -180 deg; joints [-137.467, 70.777, -83.268, 136.783, 80.829, 8.517]
  Call Extruder(789.45369)
  MoveL 9215 to (-21.1, 165.03, 125.68) mm, rotated rx -180 ry 0 rz -180 deg; joints [-137.659, 70.832, -83.215, 136.987, 80.88, 8.412]
  MoveL 9216 to (-21.1, 165.03, 125.68) mm, rotated rx -180 ry 0 rz -180 deg; joints [-137.659, 70.832, -83.215, 136.987, 80.88, 8.412]
  Call Extruder(789.88798)
  MoveL 9217 to (-21.97, 164.98, 125.68) mm, rotated rx -180 ry 0 rz 180 deg; joints [-137.804, 70.873, -83.175, 137.141, 80.918, 8.333]
  MoveL 9218 to (-21.97, 164.98, 125.68) mm, rotated rx -180 ry 0 rz 180 deg; joints [-137.804, 70.873, -83.175, 137.141, 80.918, 8.333]
  Call Extruder(790.18201)
  MoveL 9219 to (-22.56, 164.93, 125.68) mm, rotated rx 180 ry 0 rz 180 deg; joints [-137.905, 70.9, -83.149, 137.248, 80.943, 8.28]
  MoveL 9220 to (-22.56, 164.93, 125.68) mm, rotated rx 180 ry 0 rz 180 deg; joints [-137.905, 70.9, -83.149, 137.248, 80.943, 8.28]
  Call Extruder(790.47737)
  MoveL 9221 to (-23.15, 164.89, 125.68) mm, rotated rx 180 ry 0 rz -180 deg; joints [-138.004, 70.927, -83.122, 137.353, 80.967, 8.228]
  MoveL 9222 to (-23.15, 164.89, 125.68) mm, rotated rx 180 ry 0 rz -180 deg; joints [-138.004, 70.927, -83.122, 137.353, 80.967, 8.228]
  Call Extruder(790.72359)
  MoveL 9223 to (-23.64, 164.84, 125.68) mm, rotated rx 180 ry 0 rz 180 deg; joints [-138.088, 70.949, -83.101, 137.442, 80.988, 8.185]
  MoveL 9224 to (-23.64, 164.84, 125.68) mm, rotated rx 180 ry 0 rz 180 deg; joints [-138.088, 70.949, -83.101, 137.442, 80.988, 8.185]
  Call Extruder(790.92030)
  MoveL 9225 to (-24.03, 164.79, 125.68) mm, rotated rx -180 ry 0 rz -180 deg; joints [-138.156, 70.966, -83.084, 137.514, 81.003, 8.151]
  MoveL 9226 to (-24.03, 164.79, 125.68) mm, rotated rx -180 ry 0 rz -180 deg; joints [-138.156, 70.966, -83.084, 137.514, 81.003, 8.151]
  Call Extruder(791.11787)
  MoveL 9227 to (-24.42, 164.75, 125.68) mm, rotated rx 180 ry 0 rz 180 deg; joints [-138.224, 70.983, -83.067, 137.585, 81.018, 8.117]
  MoveL 9228 to (-24.42, 164.75, 125.68) mm, rotated rx 180 ry 0 rz 180 deg; joints [-138.224, 70.983, -83.067, 137.585, 81.018, 8.117]
  Call Extruder(791.31631)
  MoveL 9229 to (-24.8, 164.7, 125.68) mm, rotated rx -180 ry 0 rz -180 deg; joints [-138.292, 71, -83.05, 137.657, 81.034, 8.084]
  MoveL 9230 to (-24.8, 164.7, 125.68) mm, rotated rx -180 ry 0 rz -180 deg; joints [-138.292, 71, -83.05, 137.657, 81.034, 8.084]
  Call Extruder(791.51562)
  MoveL 9231 to (-25.19, 164.66, 125.68) mm, rotated rx -180 ry 0 rz 180 deg; joints [-138.359, 71.017, -83.033, 137.728, 81.049, 8.05]
  MoveL 9232 to (-25.19, 164.66, 125.68) mm, rotated rx -180 ry 0 rz 180 deg; joints [-138.359, 71.017, -83.033, 137.728, 81.049, 8.05]
  Call Extruder(791.67445)
  MoveL 9233 to (-25.5, 164.61, 125.68) mm, rotated rx -180 ry 0 rz 180 deg; joints [-138.415, 71.03, -83.02, 137.786, 81.061, 8.024]
  MoveL 9234 to (-25.5, 164.61, 125.68) mm, rotated rx -180 ry 0 rz 180 deg; joints [-138.415, 71.03, -83.02, 137.786, 81.061, 8.024]
  Call Extruder(791.83401)
  MoveL 9235 to (-25.8, 164.56, 125.68) mm, rotated rx 180 ry 0 rz -180 deg; joints [-138.47, 71.042, -83.007, 137.844, 81.072, 7.998]
  MoveL 9236 to (-25.8, 164.56, 125.68) mm, rotated rx 180 ry 0 rz -180 deg; joints [-138.47, 71.042, -83.007, 137.844, 81.072, 7.998]
  Call Extruder(791.99430)
  MoveL 9237 to (-26.11, 164.51, 125.68) mm, rotated rx -180 ry 0 rz 180 deg; joints [-138.525, 71.055, -82.994, 137.902, 81.084, 7.972]
  MoveL 9238 to (-26.11, 164.51, 125.68) mm, rotated rx -180 ry 0 rz 180 deg; joints [-138.525, 71.055, -82.994, 137.902, 81.084, 7.972]
  Call Extruder(792.15531)
  MoveL 9239 to (-26.41, 164.46, 125.68) mm, rotated rx -180 ry 0 rz -180 deg; joints [-138.58, 71.068, -82.981, 137.96, 81.095, 7.946]
  MoveL 9240 to (-26.41, 164.46, 125.68) mm, rotated rx -180 ry 0 rz -180 deg; joints [-138.58, 71.068, -82.981, 137.96, 81.095, 7.946]
  Call Extruder(792.31706)
  MoveL 9241 to (-26.72, 164.41, 125.68) mm, rotated rx -180 ry 0 rz -180 deg; joints [-138.635, 71.081, -82.968, 138.018, 81.107, 7.919]
  MoveL 9242 to (-26.72, 164.41, 125.68) mm, rotated rx -180 ry 0 rz -180 deg; joints [-138.635, 71.081, -82.968, 138.018, 81.107, 7.919]
  Call Extruder(792.47953)
  MoveL 9243 to (-27.02, 164.37, 125.68) mm, rotated rx -180 ry 0 rz -180 deg; joints [-138.69, 71.094, -82.955, 138.076, 81.119, 7.893]
  MoveL 9244 to (-27.02, 164.37, 125.68) mm, rotated rx -180 ry 0 rz -180 deg; joints [-138.69, 71.094, -82.955, 138.076, 81.119, 7.893]
  Call Extruder(792.61345)
  MoveL 9245 to (-27.27, 164.32, 125.68) mm, rotated rx -180 ry 0 rz 180 deg; joints [-138.736, 71.104, -82.945, 138.124, 81.127, 7.872]
  MoveL 9246 to (-27.27, 164.32, 125.68) mm, rotated rx -180 ry 0 rz 180 deg; joints [-138.736, 71.104, -82.945, 138.124, 81.127, 7.872]
  Call Extruder(792.74799)
  MoveL 9247 to (-27.52, 164.27, 125.68) mm, rotated rx 180 ry 0 rz -180 deg; joints [-138.783, 71.114, -82.934, 138.173, 81.136, 7.852]
  MoveL 9248 to (-27.52, 164.27, 125.68) mm, rotated rx 180 ry 0 rz -180 deg; joints [-138.783, 71.114, -82.934, 138.173, 81.136, 7.852]
  Call Extruder(792.88314)
  MoveL 9249 to (-27.77, 164.22, 125.68) mm, rotated rx -180 ry 0 rz 180 deg; joints [-138.829, 71.124, -82.924, 138.222, 81.145, 7.831]
  MoveL 9250 to (-27.77, 164.22, 125.68) mm, rotated rx -180 ry 0 rz 180 deg; joints [-138.829, 71.124, -82.924, 138.222, 81.145, 7.831]
  Call Extruder(793.01889)
  MoveL 9251 to (-28.02, 164.17, 125.68) mm, rotated rx -180 ry 0 rz 180 deg; joints [-138.875, 71.134, -82.914, 138.27, 81.154, 7.81]
  MoveL 9252 to (-28.02, 164.17, 125.68) mm, rotated rx -180 ry 0 rz 180 deg; joints [-138.875, 71.134, -82.914, 138.27, 81.154, 7.81]
  Call Extruder(793.15526)
  MoveL 9253 to (-28.27, 164.12, 125.68) mm, rotated rx -180 ry 0 rz -180 deg; joints [-138.921, 71.144, -82.904, 138.318, 81.163, 7.789]
  MoveL 9254 to (-28.27, 164.12, 125.68) mm, rotated rx -180 ry 0 rz -180 deg; joints [-138.921, 71.144, -82.904, 138.318, 81.163, 7.789]
  Call Extruder(793.24012)
  MoveL 9255 to (-28.43, 164.09, 125.68) mm, rotated rx 180 ry 0 rz -180 deg; joints [-138.95, 71.15, -82.897, 138.348, 81.168, 7.776]
  Set speed (130.0 mm/s)
  MoveL 9256 to (-31.76, 163.31, 125.68) mm, rotated rx -180 ry 0 rz 180 deg; joints [-139.581, 71.281, -82.762, 139.008, 81.283, 7.503]
  MoveL 9257 to (-31.76, 163.31, 135.08) mm, rotated rx 180 ry 0 rz 180 deg; joints [-139.581, 72.635, -84.521, 138.967, 80.978, 7.771]
  Call Extruder(791.24012)
  Set speed (40.0 mm/s)
  MoveL 9258 to (-31.76, 163.31, 135.08) mm, rotated rx 180 ry 0 rz 180 deg; joints [-139.581, 72.635, -84.521, 138.967, 80.978, 7.771]
  Call Extruder(0.00000)
  Set speed (130.0 mm/s)
  MoveL 9259 to (-39.41, 155.44, 135.08) mm, rotated rx 180 ry 0 rz 180 deg; joints [-142.064, 72.697, -84.456, 141.473, 80.75, 7.293]
  Call Extruder(2.00000)
  Set speed (40.0 mm/s)
  MoveL 9260 to (-39.41, 155.44, 135.08) mm, rotated rx 180 ry 0 rz 180 deg; joints [-142.064, 72.697, -84.456, 141.473, 80.75, 7.293]
  Set speed (30.0 mm/s)
  MoveL 9261 to (-39.41, 155.44, 135.08) mm, rotated rx 180 ry 0 rz 180 deg; joints [-142.064, 72.697, -84.456, 141.473, 80.75, 7.293]
  Call Extruder(2.05684)
  MoveL 9262 to (-39.44, 155.34, 135.08) mm, rotated rx 180 ry 0 rz 180 deg; joints [-142.085, 72.695, -84.459, 141.494, 80.744, 7.293]
  MoveL 9263 to (-39.44, 155.34, 135.08) mm, rotated rx 180 ry 0 rz 180 deg; joints [-142.085, 72.695, -84.459, 141.494, 80.744, 7.293]
  Call Extruder(2.17007)
  MoveL 9264 to (-39.5, 155.15, 135.08) mm, rotated rx 180 ry 0 rz 180 deg; joints [-142.127, 72.691, -84.463, 141.535, 80.732, 7.291]
  MoveL 9265 to (-39.5, 155.15, 135.08) mm, rotated rx 180 ry 0 rz 180 deg; joints [-142.127, 72.691, -84.463, 141.535, 80.732, 7.291]
  Call Extruder(2.28286)
  MoveL 9266 to (-39.56, 154.97, 135.08) mm, rotated rx -180 ry 0 rz 180 deg; joints [-142.169, 72.686, -84.468, 141.577, 80.719, 7.29]
  MoveL 9267 to (-39.56, 154.97, 135.08) mm, rotated rx -180 ry 0 rz 180 deg; joints [-142.169, 72.686, -84.468, 141.577, 80.719, 7.29]
  Call Extruder(2.39521)
  MoveL 9268 to (-39.62, 154.78, 135.08) mm, rotated rx -180 ry 0 rz 180 deg; joints [-142.212, 72.682, -84.472, 141.618, 80.707, 7.289]
  MoveL 9269 to (-39.62, 154.78, 135.08) mm, rotated rx -180 ry 0 rz 180 deg; joints [-142.212, 72.682, -84.472, 141.618, 80.707, 7.289]
  Call Extruder(2.50711)
  MoveL 9270 to (-39.68, 154.59, 135.08) mm, rotated rx -180 ry 0 rz -180 deg; joints [-142.254, 72.677, -84.477, 141.66, 80.695, 7.288]
  MoveL 9271 to (-39.68, 154.59, 135.08) mm, rotated rx -180 ry 0 rz -180 deg; joints [-142.254, 72.677, -84.477, 141.66, 80.695, 7.288]
  Call Extruder(2.62851)
  MoveL 9272 to (-39.75, 154.38, 135.08) mm, rotated rx 180 ry 0 rz 180 deg; joints [-142.3, 72.673, -84.482, 141.705, 80.681, 7.286]
  MoveL 9273 to (-39.75, 154.38, 135.08) mm, rotated rx 180 ry 0 rz 180 deg; joints [-142.3, 72.673, -84.482, 141.705, 80.681, 7.286]
  Call Extruder(2.75930)
  MoveL 9274 to (-39.81, 154.16, 135.08) mm, rotated rx -180 ry 0 rz 180 deg; joints [-142.35, 72.667, -84.488, 141.754, 80.666, 7.285]
  MoveL 9275 to (-39.81, 154.16, 135.08) mm, rotated rx -180 ry 0 rz 180 deg; joints [-142.35, 72.667, -84.488, 141.754, 80.666, 7.285]
  Call Extruder(2.88953)
  MoveL 9276 to (-39.88, 153.94, 135.08) mm, rotated rx -180 ry 0 rz -180 deg; joints [-142.399, 72.662, -84.493, 141.803, 80.651, 7.284]
  MoveL 9277 to (-39.88, 153.94, 135.08) mm, rotated rx -180 ry 0 rz -180 deg; joints [-142.399, 72.662, -84.493, 141.803, 80.651, 7.284]
  Call Extruder(3.01920)
  MoveL 9278 to (-39.95, 153.71, 135.08) mm, rotated rx -180 ry 0 rz -180 deg; joints [-142.449, 72.656, -84.499, 141.851, 80.636, 7.283]
  MoveL 9279 to (-39.95, 153.71, 135.08) mm, rotated rx -180 ry 0 rz -180 deg; joints [-142.449, 72.656, -84.499, 141.851, 80.636, 7.283]
  Call Extruder(3.14830)
  MoveL 9280 to (-40.02, 153.49, 135.08) mm, rotated rx -180 ry 0 rz -180 deg; joints [-142.498, 72.651, -84.505, 141.9, 80.621, 7.282]
  MoveL 9281 to (-40.02, 153.49, 135.08) mm, rotated rx -180 ry 0 rz -180 deg; joints [-142.498, 72.651, -84.505, 141.9, 80.621, 7.282]
  Call Extruder(3.26338)
  MoveL 9282 to (-40.06, 153.28, 135.08) mm, rotated rx -180 ry 0 rz 180 deg; joints [-142.541, 72.645, -84.51, 141.942, 80.607, 7.282]
  MoveL 9283 to (-40.06, 153.28, 135.08) mm, rotated rx -180 ry 0 rz 180 deg; joints [-142.541, 72.645, -84.51, 141.942, 80.607, 7.282]
  Call Extruder(3.37800)
  MoveL 9284 to (-40.11, 153.08, 135.08) mm, rotated rx 180 ry 0 rz -180 deg; joints [-142.584, 72.639, -84.516, 141.984, 80.592, 7.282]
  MoveL 9285 to (-40.11, 153.08, 135.08) mm, rotated rx 180 ry 0 rz -180 deg; joints [-142.584, 72.639, -84.516, 141.984, 80.592, 7.282]
  Call Extruder(3.49217)
  MoveL 9286 to (-40.15, 152.88, 135.08) mm, rotated rx -180 ry 0 rz -180 deg; joints [-142.627, 72.634, -84.522, 142.026, 80.577, 7.282]
  MoveL 9287 to (-40.15, 152.88, 135.08) mm, rotated rx -180 ry 0 rz -180 deg; joints [-142.627, 72.634, -84.522, 142.026, 80.577, 7.282]
  Call Extruder(3.60589)
  MoveL 9288 to (-40.2, 152.67, 135.08) mm, rotated rx -180 ry 0 rz 180 deg; joints [-142.671, 72.628, -84.528, 142.069, 80.562, 7.283]
  MoveL 9289 to (-40.2, 152.67, 135.08) mm, rotated rx -180 ry 0 rz 180 deg; joints [-142.671, 72.628, -84.528, 142.069, 80.562, 7.283]
  Call Extruder(3.70891)
  MoveL 9290 to (-40.24, 152.49, 135.08) mm, rotated rx 180 ry 0 rz -180 deg; joints [-142.71, 72.622, -84.534, 142.107, 80.549, 7.283]
  MoveL 9291 to (-40.24, 152.49, 135.08) mm, rotated rx 180 ry 0 rz -180 deg; joints [-142.71, 72.622, -84.534, 142.107, 80.549, 7.283]
  Call Extruder(3.80140)
  MoveL 9292 to (-40.27, 152.32, 135.08) mm, rotated rx -180 ry 0 rz -180 deg; joints [-142.745, 72.617, -84.539, 142.141, 80.536, 7.283]
  Set speed (130.0 mm/s)
  MoveL 9293 to (-40.27, 152.32, 135.08) mm, rotated rx -180 ry 0 rz -180 deg; joints [-142.745, 72.617, -84.539, 142.141, 80.536, 7.283]
  Set speed (30.0 mm/s)
  MoveL 9294 to (-40.27, 152.32, 135.08) mm, rotated rx -180 ry 0 rz -180 deg; joints [-142.745, 72.617, -84.539, 142.141, 80.536, 7.283]
  Call Extruder(3.93780)
  MoveL 9295 to (-40.32, 152.07, 135.08) mm, rotated rx -180 ry 0 rz 180 deg; joints [-142.796, 72.61, -84.546, 142.192, 80.518, 7.284]
  MoveL 9296 to (-40.32, 152.07, 135.08) mm, rotated rx -180 ry 0 rz 180 deg; joints [-142.796, 72.61, -84.546, 142.192, 80.518, 7.284]
  Call Extruder(4.07360)
  MoveL 9297 to (-40.37, 151.82, 135.08) mm, rotated rx 180 ry 0 rz 180 deg; joints [-142.848, 72.603, -84.554, 142.242, 80.5, 7.285]
  MoveL 9298 to (-40.37, 151.82, 135.08) mm, rotated rx 180 ry 0 rz 180 deg; joints [-142.848, 72.603, -84.554, 142.242, 80.5, 7.285]
  Call Extruder(4.20879)
  MoveL 9299 to (-40.42, 151.57, 135.08) mm, rotated rx -180 ry 0 rz -180 deg; joints [-142.901, 72.596, -84.561, 142.293, 80.482, 7.285]
  MoveL 9300 to (-40.42, 151.57, 135.08) mm, rotated rx -180 ry 0 rz -180 deg; joints [-142.901, 72.596, -84.561, 142.293, 80.482, 7.285]
  Call Extruder(4.34337)
  MoveL 9301 to (-40.47, 151.32, 135.08) mm, rotated rx -180 ry 0 rz -180 deg; joints [-142.952, 72.588, -84.569, 142.344, 80.464, 7.285]
  MoveL 9302 to (-40.47, 151.32, 135.08) mm, rotated rx -180 ry 0 rz -180 deg; joints [-142.952, 72.588, -84.569, 142.344, 80.464, 7.285]
  Call Extruder(4.47734)
  MoveL 9303 to (-40.52, 151.07, 135.08) mm, rotated rx -180 ry 0 rz 180 deg; joints [-143.005, 72.581, -84.576, 142.395, 80.445, 7.286]
  MoveL 9304 to (-40.52, 151.07, 135.08) mm, rotated rx -180 ry 0 rz 180 deg; joints [-143.005, 72.581, -84.576, 142.395, 80.445, 7.286]
  Call Extruder(4.61071)
  MoveL 9305 to (-40.56, 150.82, 135.08) mm, rotated rx 180 ry 0 rz 180 deg; joints [-143.057, 72.574, -84.584, 142.446, 80.427, 7.286]
  MoveL 9306 to (-40.56, 150.82, 135.08) mm, rotated rx 180 ry 0 rz 180 deg; joints [-143.057, 72.574, -84.584, 142.446, 80.427, 7.286]
  Call Extruder(4.77280)
  MoveL 9307 to (-40.61, 150.52, 135.08) mm, rotated rx -180 ry 0 rz 180 deg; joints [-143.119, 72.564, -84.593, 142.507, 80.404, 7.287]
  MoveL 9308 to (-40.61, 150.52, 135.08) mm, rotated rx -180 ry 0 rz 180 deg; joints [-143.119, 72.564, -84.593, 142.507, 80.404, 7.287]
  Call Extruder(4.93416)
  MoveL 9309 to (-40.66, 150.21, 135.08) mm, rotated rx -180 ry 0 rz 180 deg; joints [-143.182, 72.555, -84.603, 142.568, 80.381, 7.289]
  MoveL 9310 to (-40.66, 150.21, 135.08) mm, rotated rx -180 ry 0 rz 180 deg; joints [-143.182, 72.555, -84.603, 142.568, 80.381, 7.289]
  Call Extruder(5.09479)
  MoveL 9311 to (-40.71, 149.91, 135.08) mm, rotated rx 180 ry 0 rz 180 deg; joints [-143.245, 72.545, -84.613, 142.629, 80.358, 7.29]
  MoveL 9312 to (-40.71, 149.91, 135.08) mm, rotated rx 180 ry 0 rz 180 deg; joints [-143.245, 72.545, -84.613, 142.629, 80.358, 7.29]
  Call Extruder(5.25470)
  MoveL 9313 to (-40.76, 149.6, 135.08) mm, rotated rx 180 ry 0 rz 180 deg; joints [-143.307, 72.536, -84.622, 142.69, 80.335, 7.291]
  MoveL 9314 to (-40.76, 149.6, 135.08) mm, rotated rx 180 ry 0 rz 180 deg; joints [-143.307, 72.536, -84.622, 142.69, 80.335, 7.291]
  Call Extruder(5.41388)
  MoveL 9315 to (-40.81, 149.3, 135.08) mm, rotated rx -180 ry 0 rz 180 deg; joints [-143.37, 72.527, -84.632, 142.751, 80.311, 7.292]
  MoveL 9316 to (-40.81, 149.3, 135.08) mm, rotated rx -180 ry 0 rz 180 deg; joints [-143.37, 72.527, -84.632, 142.751, 80.311, 7.292]
  Call Extruder(5.57233)
  MoveL 9317 to (-40.86, 148.99, 135.08) mm, rotated rx 180 ry 0 rz 180 deg; joints [-143.433, 72.517, -84.641, 142.812, 80.288, 7.293]
  MoveL 9318 to (-40.86, 148.99, 135.08) mm, rotated rx 180 ry 0 rz 180 deg; joints [-143.433, 72.517, -84.641, 142.812, 80.288, 7.293]
  Call Extruder(5.77120)
  MoveL 9319 to (-40.9, 148.6, 135.08) mm, rotated rx -180 ry 0 rz 180 deg; joints [-143.51, 72.504, -84.654, 142.888, 80.258, 7.296]
  MoveL 9320 to (-40.9, 148.6, 135.08) mm, rotated rx -180 ry 0 rz 180 deg; joints [-143.51, 72.504, -84.654, 142.888, 80.258, 7.296]
  Call Extruder(5.96921)
  MoveL 9321 to (-40.95, 148.22, 135.08) mm, rotated rx -180 ry 0 rz -180 deg; joints [-143.588, 72.491, -84.667, 142.963, 80.228, 7.298]
  MoveL 9322 to (-40.95, 148.22, 135.08) mm, rotated rx -180 ry 0 rz -180 deg; joints [-143.588, 72.491, -84.667, 142.963, 80.228, 7.298]
  Call Extruder(6.16635)
  MoveL 9323 to (-40.99, 147.83, 135.08) mm, rotated rx -180 ry 0 rz 180 deg; joints [-143.666, 72.479, -84.68, 143.039, 80.197, 7.301]
  MoveL 9324 to (-40.99, 147.83, 135.08) mm, rotated rx -180 ry 0 rz 180 deg; joints [-143.666, 72.479, -84.68, 143.039, 80.197, 7.301]
  Call Extruder(6.36262)
  MoveL 9325 to (-41.04, 147.44, 135.08) mm, rotated rx -180 ry 0 rz -180 deg; joints [-143.744, 72.466, -84.693, 143.115, 80.167, 7.303]
  MoveL 9326 to (-41.04, 147.44, 135.08) mm, rotated rx -180 ry 0 rz -180 deg; joints [-143.744, 72.466, -84.693, 143.115, 80.167, 7.303]
  Call Extruder(6.60831)
  MoveL 9327 to (-41.09, 146.95, 135.08) mm, rotated rx -180 ry 0 rz 180 deg; joints [-143.841, 72.449, -84.71, 143.209, 80.128, 7.306]
  MoveL 9328 to (-41.09, 146.95, 135.08) mm, rotated rx -180 ry 0 rz 180 deg; joints [-143.841, 72.449, -84.71, 143.209, 80.128, 7.306]
  Call Extruder(6.90304)
  MoveL 9329 to (-41.13, 146.36, 135.08) mm, rotated rx -180 ry 0 rz 180 deg; joints [-143.957, 72.429, -84.73, 143.321, 80.08, 7.311]
  MoveL 9330 to (-41.13, 146.36, 135.08) mm, rotated rx -180 ry 0 rz 180 deg; joints [-143.957, 72.429, -84.73, 143.321, 80.08, 7.311]
  Call Extruder(7.19644)
  MoveL 9331 to (-41.18, 145.77, 135.08) mm, rotated rx -180 ry 0 rz -180 deg; joints [-144.073, 72.408, -84.751, 143.434, 80.033, 7.316]
  MoveL 9332 to (-41.18, 145.77, 135.08) mm, rotated rx -180 ry 0 rz -180 deg; joints [-144.073, 72.408, -84.751, 143.434, 80.033, 7.316]
  Call Extruder(7.62977)
  MoveL 9333 to (-41.23, 144.9, 135.08) mm, rotated rx 180 ry 0 rz -180 deg; joints [-144.243, 72.377, -84.782, 143.599, 79.96, 7.324]
  MoveL 9334 to (-41.23, 144.9, 135.08) mm, rotated rx 180 ry 0 rz -180 deg; joints [-144.243, 72.377, -84.782, 143.599, 79.96, 7.324]
  Call Extruder(8.20193)
  MoveL 9335 to (-41.27, 143.74, 135.08) mm, rotated rx 180 ry 0 rz -180 deg; joints [-144.468, 72.334, -84.824, 143.816, 79.863, 7.336]
  MoveL 9336 to (-41.27, 143.74, 135.08) mm, rotated rx 180 ry 0 rz -180 deg; joints [-144.468, 72.334, -84.824, 143.816, 79.863, 7.336]
  Call Extruder(8.62976)
  MoveL 9337 to (-41.29, 142.86, 135.08) mm, rotated rx -180 ry 0 rz 180 deg; joints [-144.635, 72.301, -84.856, 143.978, 79.789, 7.345]
  Call Extruder(50.62329)
  MoveL 9338 to (-41.29, 57.14, 135.08) mm, rotated rx 180 ry 0 rz 180 deg; joints [-164.153, 69.539, -87.057, 163.423, 73.168, 4.926]
  MoveL 9339 to (-41.29, 57.14, 135.08) mm, rotated rx 180 ry 0 rz 180 deg; joints [-164.153, 69.539, -87.057, 163.423, 73.168, 4.926]
  Call Extruder(51.33886)
  MoveL 9340 to (-41.25, 55.68, 135.08) mm, rotated rx -180 ry 0 rz 180 deg; joints [-164.534, 69.505, -87.08, 163.815, 73.081, 4.828]
  MoveL 9341 to (-41.25, 55.68, 135.08) mm, rotated rx -180 ry 0 rz 180 deg; joints [-164.534, 69.505, -87.08, 163.815, 73.081, 4.828]
  Call Extruder(51.91360)
  MoveL 9342 to (-41.2, 54.52, 135.08) mm, rotated rx -180 ry 0 rz -180 deg; joints [-164.838, 69.477, -87.098, 164.129, 73.012, 4.749]
  MoveL 9343 to (-41.2, 54.52, 135.08) mm, rotated rx -180 ry 0 rz -180 deg; joints [-164.838, 69.477, -87.098, 164.129, 73.012, 4.749]
  Call Extruder(52.20698)
  MoveL 9344 to (-41.15, 53.93, 135.08) mm, rotated rx -180 ry 0 rz 180 deg; joints [-164.992, 69.461, -87.108, 164.286, 72.974, 4.709]
  MoveL 9345 to (-41.15, 53.93, 135.08) mm, rotated rx -180 ry 0 rz 180 deg; joints [-164.992, 69.461, -87.108, 164.286, 72.974, 4.709]
  Call Extruder(52.50168)
  MoveL 9346 to (-41.11, 53.34, 135.08) mm, rotated rx -180 ry 0 rz 180 deg; joints [-165.145, 69.445, -87.118, 164.444, 72.937, 4.67]
  MoveL 9347 to (-41.11, 53.34, 135.08) mm, rotated rx -180 ry 0 rz 180 deg; joints [-165.145, 69.445, -87.118, 164.444, 72.937, 4.67]
  Call Extruder(52.79772)
  MoveL 9348 to (-41.06, 52.75, 135.08) mm, rotated rx 180 ry 0 rz 180 deg; joints [-165.299, 69.43, -87.128, 164.602, 72.899, 4.63]
  MoveL 9349 to (-41.06, 52.75, 135.08) mm, rotated rx 180 ry 0 rz 180 deg; joints [-165.299, 69.43, -87.128, 164.602, 72.899, 4.63]
  Call Extruder(52.99180)
  MoveL 9350 to (-41.02, 52.37, 135.08) mm, rotated rx -180 ry 0 rz -180 deg; joints [-165.398, 69.418, -87.135, 164.704, 72.874, 4.605]
  MoveL 9351 to (-41.02, 52.37, 135.08) mm, rotated rx -180 ry 0 rz -180 deg; joints [-165.398, 69.418, -87.135, 164.704, 72.874, 4.605]
  Call Extruder(53.18958)
  MoveL 9352 to (-40.97, 51.98, 135.08) mm, rotated rx -180 ry 0 rz 180 deg; joints [-165.498, 69.407, -87.142, 164.807, 72.848, 4.579]
  MoveL 9353 to (-40.97, 51.98, 135.08) mm, rotated rx -180 ry 0 rz 180 deg; joints [-165.498, 69.407, -87.142, 164.807, 72.848, 4.579]
  Call Extruder(53.38824)
  MoveL 9354 to (-40.92, 51.59, 135.08) mm, rotated rx -180 ry 0 rz -180 deg; joints [-165.599, 69.396, -87.149, 164.911, 72.822, 4.553]
  MoveL 9355 to (-40.92, 51.59, 135.08) mm, rotated rx -180 ry 0 rz -180 deg; joints [-165.599, 69.396, -87.149, 164.911, 72.822, 4.553]
  Call Extruder(53.58777)
  MoveL 9356 to (-40.88, 51.2, 135.08) mm, rotated rx -180 ry 0 rz 180 deg; joints [-165.7, 69.384, -87.157, 165.015, 72.796, 4.527]
  MoveL 9357 to (-40.88, 51.2, 135.08) mm, rotated rx -180 ry 0 rz 180 deg; joints [-165.7, 69.384, -87.157, 165.015, 72.796, 4.527]
  Call Extruder(53.76717)
  MoveL 9358 to (-40.83, 50.86, 135.08) mm, rotated rx 180 ry 0 rz 180 deg; joints [-165.79, 69.374, -87.163, 165.107, 72.772, 4.504]
  MoveL 9359 to (-40.83, 50.86, 135.08) mm, rotated rx 180 ry 0 rz 180 deg; joints [-165.79, 69.374, -87.163, 165.107, 72.772, 4.504]
  Call Extruder(53.92635)
  MoveL 9360 to (-40.78, 50.55, 135.08) mm, rotated rx -180 ry 0 rz 180 deg; joints [-165.869, 69.364, -87.169, 165.188, 72.751, 4.484]
  MoveL 9361 to (-40.78, 50.55, 135.08) mm, rotated rx -180 ry 0 rz 180 deg; joints [-165.869, 69.364, -87.169, 165.188, 72.751, 4.484]
  Call Extruder(54.08625)
  MoveL 9362 to (-40.73, 50.24, 135.08) mm, rotated rx 180 ry 0 rz 180 deg; joints [-165.948, 69.354, -87.176, 165.269, 72.729, 4.463]
  MoveL 9363 to (-40.73, 50.24, 135.08) mm, rotated rx 180 ry 0 rz 180 deg; joints [-165.948, 69.354, -87.176, 165.269, 72.729, 4.463]
  Call Extruder(54.24689)
  MoveL 9364 to (-40.69, 49.94, 135.08) mm, rotated rx -180 ry 0 rz -180 deg; joints [-166.026, 69.344, -87.182, 165.35, 72.708, 4.443]
  MoveL 9365 to (-40.69, 49.94, 135.08) mm, rotated rx -180 ry 0 rz -180 deg; joints [-166.026, 69.344, -87.182, 165.35, 72.708, 4.443]
  Call Extruder(54.40825)
  MoveL 9366 to (-40.64, 49.63, 135.08) mm, rotated rx 180 ry 0 rz -180 deg; joints [-166.105, 69.335, -87.188, 165.432, 72.686, 4.423]
  MoveL 9367 to (-40.64, 49.63, 135.08) mm, rotated rx 180 ry 0 rz -180 deg; joints [-166.105, 69.335, -87.188, 165.432, 72.686, 4.423]
  Call Extruder(54.57034)
  MoveL 9368 to (-40.59, 49.33, 135.08) mm, rotated rx -180 ry 0 rz -180 deg; joints [-166.184, 69.325, -87.194, 165.513, 72.665, 4.402]
  MoveL 9369 to (-40.59, 49.33, 135.08) mm, rotated rx -180 ry 0 rz -180 deg; joints [-166.184, 69.325, -87.194, 165.513, 72.665, 4.402]
  Call Extruder(54.71853)
  MoveL 9370 to (-40.54, 49.05, 135.08) mm, rotated rx -180 ry 0 rz 180 deg; joints [-166.256, 69.316, -87.2, 165.586, 72.645, 4.384]
  MoveL 9371 to (-40.54, 49.05, 135.08) mm, rotated rx -180 ry 0 rz 180 deg; joints [-166.256, 69.316, -87.2, 165.586, 72.645, 4.384]
  Call Extruder(54.85276)
  MoveL 9372 to (-40.49, 48.8, 135.08) mm, rotated rx -180 ry 0 rz 180 deg; joints [-166.32, 69.307, -87.205, 165.652, 72.626, 4.368]
  MoveL 9373 to (-40.49, 48.8, 135.08) mm, rotated rx -180 ry 0 rz 180 deg; joints [-166.32, 69.307, -87.205, 165.652, 72.626, 4.368]
  Call Extruder(54.98760)
  MoveL 9374 to (-40.44, 48.55, 135.08) mm, rotated rx 180 ry 0 rz 180 deg; joints [-166.384, 69.299, -87.21, 165.718, 72.608, 4.351]
  MoveL 9375 to (-40.44, 48.55, 135.08) mm, rotated rx 180 ry 0 rz 180 deg; joints [-166.384, 69.299, -87.21, 165.718, 72.608, 4.351]
  Call Extruder(55.12305)
  MoveL 9376 to (-40.39, 48.3, 135.08) mm, rotated rx -180 ry 0 rz 180 deg; joints [-166.448, 69.29, -87.216, 165.784, 72.59, 4.335]
  MoveL 9377 to (-40.39, 48.3, 135.08) mm, rotated rx -180 ry 0 rz 180 deg; joints [-166.448, 69.29, -87.216, 165.784, 72.59, 4.335]
  Call Extruder(55.25911)
  MoveL 9378 to (-40.34, 48.05, 135.08) mm, rotated rx -180 ry 0 rz 180 deg; joints [-166.512, 69.281, -87.221, 165.85, 72.571, 4.318]
  MoveL 9379 to (-40.34, 48.05, 135.08) mm, rotated rx -180 ry 0 rz 180 deg; joints [-166.512, 69.281, -87.221, 165.85, 72.571, 4.318]
  Call Extruder(55.39578)
  MoveL 9380 to (-40.29, 47.8, 135.08) mm, rotated rx 180 ry 0 rz 180 deg; joints [-166.576, 69.273, -87.226, 165.916, 72.553, 4.302]
  MoveL 9381 to (-40.29, 47.8, 135.08) mm, rotated rx 180 ry 0 rz 180 deg; joints [-166.576, 69.273, -87.226, 165.916, 72.553, 4.302]
  Call Extruder(55.53306)
  MoveL 9382 to (-40.24, 47.56, 135.08) mm, rotated rx -180 ry 0 rz 180 deg; joints [-166.641, 69.264, -87.232, 165.982, 72.535, 4.285]
  MoveL 9383 to (-40.24, 47.56, 135.08) mm, rotated rx -180 ry 0 rz 180 deg; joints [-166.641, 69.264, -87.232, 165.982, 72.535, 4.285]
  Call Extruder(55.65874)
  MoveL 9384 to (-40.2, 47.33, 135.08) mm, rotated rx -180 ry 0 rz 180 deg; joints [-166.699, 69.256, -87.237, 166.042, 72.518, 4.27]
  MoveL 9385 to (-40.2, 47.33, 135.08) mm, rotated rx -180 ry 0 rz 180 deg; joints [-166.699, 69.256, -87.237, 166.042, 72.518, 4.27]
  Call Extruder(55.77269)
  MoveL 9386 to (-40.15, 47.12, 135.08) mm, rotated rx 180 ry 0 rz 180 deg; joints [-166.751, 69.249, -87.241, 166.096, 72.502, 4.257]
  MoveL 9387 to (-40.15, 47.12, 135.08) mm, rotated rx 180 ry 0 rz 180 deg; joints [-166.751, 69.249, -87.241, 166.096, 72.502, 4.257]
  Call Extruder(55.88710)
  MoveL 9388 to (-40.11, 46.92, 135.08) mm, rotated rx -180 ry 0 rz -180 deg; joints [-166.804, 69.242, -87.246, 166.15, 72.487, 4.243]
  MoveL 9389 to (-40.11, 46.92, 135.08) mm, rotated rx -180 ry 0 rz -180 deg; joints [-166.804, 69.242, -87.246, 166.15, 72.487, 4.243]
  Call Extruder(56.00196)
  MoveL 9390 to (-40.06, 46.72, 135.08) mm, rotated rx 180 ry 0 rz -180 deg; joints [-166.857, 69.234, -87.25, 166.204, 72.472, 4.229]
  MoveL 9391 to (-40.06, 46.72, 135.08) mm, rotated rx 180 ry 0 rz -180 deg; joints [-166.857, 69.234, -87.25, 166.204, 72.472, 4.229]
  Call Extruder(56.11727)
  MoveL 9392 to (-40.02, 46.51, 135.08) mm, rotated rx 180 ry 0 rz -180 deg; joints [-166.909, 69.227, -87.255, 166.258, 72.456, 4.216]
  MoveL 9393 to (-40.02, 46.51, 135.08) mm, rotated rx 180 ry 0 rz -180 deg; joints [-166.909, 69.227, -87.255, 166.258, 72.456, 4.216]
  Call Extruder(56.24665)
  MoveL 9394 to (-39.95, 46.29, 135.08) mm, rotated rx 180 ry 0 rz 180 deg; joints [-166.966, 69.218, -87.261, 166.316, 72.437, 4.202]
  MoveL 9395 to (-39.95, 46.29, 135.08) mm, rotated rx 180 ry 0 rz 180 deg; joints [-166.966, 69.218, -87.261, 166.316, 72.437, 4.202]
  Call Extruder(56.37660)
  MoveL 9396 to (-39.88, 46.06, 135.08) mm, rotated rx -180 ry 0 rz 180 deg; joints [-167.022, 69.208, -87.266, 166.375, 72.418, 4.188]
  MoveL 9397 to (-39.88, 46.06, 135.08) mm, rotated rx -180 ry 0 rz 180 deg; joints [-167.022, 69.208, -87.266, 166.375, 72.418, 4.188]
  Call Extruder(56.50711)
  MoveL 9398 to (-39.82, 45.84, 135.08) mm, rotated rx 180 ry 0 rz -180 deg; joints [-167.079, 69.199, -87.272, 166.433, 72.4, 4.174]
  MoveL 9399 to (-39.82, 45.84, 135.08) mm, rotated rx 180 ry 0 rz -180 deg; joints [-167.079, 69.199, -87.272, 166.433, 72.4, 4.174]
  Call Extruder(56.63818)
  MoveL 9400 to (-39.75, 45.62, 135.08) mm, rotated rx 180 ry 0 rz 180 deg; joints [-167.136, 69.19, -87.278, 166.491, 72.381, 4.159]
  MoveL 9401 to (-39.75, 45.62, 135.08) mm, rotated rx 180 ry 0 rz 180 deg; joints [-167.136, 69.19, -87.278, 166.491, 72.381, 4.159]
  Call Extruder(56.75983)
  MoveL 9402 to (-39.68, 45.41, 135.08) mm, rotated rx 180 ry 0 rz 180 deg; joints [-167.188, 69.181, -87.283, 166.544, 72.363, 4.146]
  MoveL 9403 to (-39.68, 45.41, 135.08) mm, rotated rx 180 ry 0 rz 180 deg; joints [-167.188, 69.181, -87.283, 166.544, 72.363, 4.146]
  Call Extruder(56.87195)
  MoveL 9404 to (-39.62, 45.22, 135.08) mm, rotated rx 180 ry 0 rz 180 deg; joints [-167.235, 69.172, -87.288, 166.593, 72.347, 4.134]
  MoveL 9405 to (-39.62, 45.22, 135.08) mm, rotated rx 180 ry 0 rz 180 deg; joints [-167.235, 69.172, -87.288, 166.593, 72.347, 4.134]
  Call Extruder(56.98452)
  MoveL 9406 to (-39.56, 45.03, 135.08) mm, rotated rx -180 ry 0 rz 180 deg; joints [-167.283, 69.164, -87.293, 166.642, 72.33, 4.122]
  MoveL 9407 to (-39.56, 45.03, 135.08) mm, rotated rx -180 ry 0 rz 180 deg; joints [-167.283, 69.164, -87.293, 166.642, 72.33, 4.122]
  Call Extruder(57.09753)
  MoveL 9408 to (-39.5, 44.85, 135.08) mm, rotated rx -180 ry 0 rz 180 deg; joints [-167.331, 69.156, -87.298, 166.691, 72.314, 4.11]
